	{attribute 'TcIecLibraryType'}
	{attribute 'external_name' := 'F_VN_GradeDataMatrixCodeExp_GUID_48B47258_A931_D3A4_9456_254A5AD23142'}
	(* Grades a Data Matrix code (ECC200) according to ISO / IEC 15415:2011. Requires uniform illumination, good focus and the image sensor plane parallel to the code plane to achieve meaningful results. (expert function) *)
	FUNCTION F_VN_GradeDataMatrixCodeExp : HRESULT
	VAR_INPUT
		ipSrcImage	:	ITcVnImage;	(* Source image, only containing the Data Matrix code region (USINT, 1 channel, including quiet zone) *)
		ipDecodedData	:	REFERENCE TO ITcVnContainer;	(* Returns the decoded data (ContainerType_String_SINT) *)
	END_VAR
	VAR_IN_OUT
		stCodeGrades	:	TcVnCodeGradesDM;	(* Returns the code grades in the range from 0 (very bad) to 4 (very good) *)
	END_VAR
	VAR_INPUT
		fModuleWidth	:	REAL;	(* Minimum module width of the code in the image (in pixels). Must be at least 3, preferably 5 - 8. *)
		ipResultVisualization	:	REFERENCE TO ITcVnImage;	(* Returns a visualization of the scan grid (optional, set to 0 if not required). Module margin grades are color coded: >= 3 as green, >= 2 as light blue, >= 1 as orange, < 1 as red *)
		ipMarginGrades	:	REFERENCE TO ITcVnContainer;	(* Returns the individual margin grade for each module, e.g. to create a custom visualization (optional, set to 0 if not required; ContainerType_Vector_TcVnVector3_REAL, containing [x-position, y-position, grade]) *)
		ipContour	:	REFERENCE TO ITcVnContainer;	(* Returns the 4 code corner points, excluding the quiet zone (optional, set to 0 if not required; ContainerType_Vector_TcVnPoint2_DINT) *)
		hrPrev	:	HRESULT;	(* HRESULT indicating the result of previous operations (If SUCCEEDED(hrPrev) equals false, no operation is executed.) *)
	END_VAR
	VAR_OUTPUT
		fAngleDeg	:	REAL;	(* Returns the clockwise rotation angle in degree *)
	END_VAR

END_FUNCTION

// Functions/Code Quality/F_VN_GradeQRCode

	{attribute 'TcIecLibraryType'}
	{attribute 'external_name' := 'F_VN_GradeQRCode_GUID_2796A0BC_8AD9_DF0A_A63B_3634863F0828'}
	(* Grades a QR code according to ISO / IEC 15415:2011. Requires uniform illumination, good focus and the image sensor plane parallel to the code plane to achieve meaningful results. *)
	FUNCTION F_VN_GradeQRCode : HRESULT
	VAR_INPUT
		ipSrcImage	:	ITcVnImage;	(* Source image, only containing the QR code region (USINT, 1 channel, including quiet zone) *)
		ipDecodedData	:	REFERENCE TO ITcVnContainer;	(* Returns the decoded data (ContainerType_String_SINT) *)
	END_VAR
	VAR_IN_OUT
		stCodeGrades	:	TcVnCodeGradesQR;	(* Returns the code grades in the range from 0 (very bad) to 4 (very good) *)
	END_VAR
	VAR_INPUT
		fModuleWidth	:	REAL;	(* Minimum module width of the code in the image (in pixels). Must be at least 3, preferably 5 - 8. *)
		hrPrev	:	HRESULT;	(* HRESULT indicating the result of previous operations (If SUCCEEDED(hrPrev) equals false, no operation is executed.) *)
	END_VAR
	VAR_OUTPUT
		fAngleDeg	:	REAL;	(* Returns the clockwise rotation angle in degree *)
	END_VAR

END_FUNCTION

// Functions/Code Quality/F_VN_GradeQRCodeExp

	{attribute 'TcIecLibraryType'}
	{attribute 'external_name' := 'F_VN_GradeQRCodeExp_GUID_748E667E_FDFB_D812_893A_DF121E555FAA'}
	(* Grades a QR code according to ISO / IEC 15415:2011. Requires uniform illumination, good focus and the image sensor plane parallel to the code plane to achieve meaningful results. (expert function) *)
	FUNCTION F_VN_GradeQRCodeExp : HRESULT
	VAR_INPUT
		ipSrcImage	:	ITcVnImage;	(* Source image, only containing the QR code region (USINT, 1 channel, including quiet zone) *)
		ipDecodedData	:	REFERENCE TO ITcVnContainer;	(* Returns the decoded data (ContainerType_String_SINT) *)
	END_VAR
	VAR_IN_OUT
		stCodeGrades	:	TcVnCodeGradesQR;	(* Returns the code grades in the range from 0 (very bad) to 4 (very good) *)
	END_VAR
	VAR_INPUT
		fModuleWidth	:	REAL;	(* Minimum module width of the code in the image (in pixels). Must be at least 3, preferably 5 - 8. *)
		ipResultVisualization	:	REFERENCE TO ITcVnImage;	(* Returns a visualization of the scan grid (optional, set to 0 if not required). Module margin grades are color coded: >= 3 as green, >= 2 as light blue, >= 1 as orange, < 1 as red *)
		ipMarginGrades	:	REFERENCE TO ITcVnContainer;	(* Returns the individual margin grade for each module, e.g. to create a custom visualization (optional, set to 0 if not required; ContainerType_Vector_TcVnVector3_REAL, containing [x-position, y-position, grade]) *)
		ipContour	:	REFERENCE TO ITcVnContainer;	(* Returns the 4 code corner points, excluding the quiet zone (optional, set to 0 if not required; ContainerType_Vector_TcVnPoint2_DINT) *)
		hrPrev	:	HRESULT;	(* HRESULT indicating the result of previous operations (If SUCCEEDED(hrPrev) equals false, no operation is executed.) *)
	END_VAR
	VAR_OUTPUT
		fAngleDeg	:	REAL;	(* Returns the clockwise rotation angle in degree *)
	END_VAR

END_FUNCTION

// Functions/Texture Analysis/F_VN_Granulometry

	{attribute 'TcIecLibraryType'}
	{attribute 'external_name' := 'F_VN_Granulometry_GUID_ED4C52B4_5143_D78F_B20E_04305B4C8FA0'}
	(* Computes the granulometry of a textured image using morphological operations. *)
	FUNCTION F_VN_Granulometry : HRESULT
	VAR_INPUT
		ipImage	:	ITcVnImage;	(* Source image (1 channel) *)
		ipIntensityDiffs	:	REFERENCE TO ITcVnContainer;	(* Returns the intensity differences between successive structuring element sizes (CTcVnContainer_Vector_LREAL), which can be used as features for texture description. *)
		eMorphType	:	ETcVnMorphologicalOperator;	(* Only opening or closing are supported. *)
		nMinSize	:	UDINT;	(* Min structuring element size (odd, >= 3) *)
		nMaxSize	:	UDINT;	(* Max structuring element size (>= nMinSize) *)
		nStep	:	UDINT;	(* Step, by which nMinSize is incremented until nMaxSize is exceeded (even, >= 2). *)
		hrPrev	:	HRESULT;	(* HRESULT indicating the result of previous operations (If SUCCEEDED(hrPrev) equals false, no operation is executed.) *)
	END_VAR

END_FUNCTION

// Functions/Texture Analysis/F_VN_HaralickFeatures

	{attribute 'TcIecLibraryType'}
	{attribute 'external_name' := 'F_VN_HaralickFeatures_GUID_C04B3742_2975_D01D_971B_239AA26ADB64'}
	(* Computes the Haralick features of a graylevel image, which describe the texture. *)
	FUNCTION F_VN_HaralickFeatures : HRESULT
	VAR_INPUT
		ipImage	:	ITcVnImage;	(* Source image (1 channel, USINT) *)
		ipFeatures	:	REFERENCE TO ITcVnContainer;	(* Returns the computed Haralick features (CTcVnContainer_Vector_LREAL). The returned feature set contains the mean and standard deviation for each of the first 13 Haralick features, computed for 0, 45, 90, 135 degrees. So there will be 26 features in total (f1 mean, f1 stdDev, f2 mean, f2 stdDev, ..., f13 mean, f13 stdDev). *)
		nDist	:	UDINT;	(* Distance *)
		hrPrev	:	HRESULT;	(* HRESULT indicating the result of previous operations (If SUCCEEDED(hrPrev) equals false, no operation is executed.) *)
	END_VAR

END_FUNCTION

// Functions/OCR/F_VN_OCR

	{attribute 'TcIecLibraryType'}
	{attribute 'external_name' := 'F_VN_OCR_GUID_4649D880_E3A0_D7D8_A83C_DD423A1D4FD0'}
	(* Detects and recognizes characters in a binary image (white characters on black background). *)
	FUNCTION F_VN_OCR : HRESULT
	VAR_INPUT
		ipSrcImage	:	ITcVnImage;	(* Source image (USINT, 1 channel, binary) *)
		eModel	:	ULINT;	(* Selection of OCR model types (ETcVnOcrModelType) *)
		ipCharacters	:	REFERENCE TO ITcVnContainer;	(* Returns the recognized characters (ContainerType_Vector_String_SINT) *)
		hrPrev	:	HRESULT;	(* HRESULT indicating the result of previous operations (If SUCCEEDED(hrPrev) equals false, no operation is executed.) *)
	END_VAR

END_FUNCTION

// Functions/OCR/F_VN_OCRExp

	{attribute 'TcIecLibraryType'}
	{attribute 'external_name' := 'F_VN_OCRExp_GUID_EDBCFF98_0425_D60E_8A16_A0CDB823D474'}
	(* Detects and recognizes characters in a binary image (white characters on black background). (expert function) *)
	FUNCTION F_VN_OCRExp : HRESULT
	VAR_INPUT
		ipSrcImage	:	ITcVnImage;	(* Source image (USINT, 1 channel, binary) *)
		eModel	:	ULINT;	(* Selection of OCR model types (ETcVnOcrModelType) *)
		ipCharacters	:	REFERENCE TO ITcVnContainer;	(* Returns the recognized characters (ContainerType_Vector_String_SINT) *)
	END_VAR
	VAR_IN_OUT CONSTANT
		sPattern	:	STRING;	(* String pattern containing the format in which characters are presented *)
	END_VAR
	VAR_INPUT
		eOcrOptions	:	UDINT;	(* Specifies which options must be applied to the function (ETcVnOcrOptions) *)
		ipBoundingBoxes	:	REFERENCE TO ITcVnContainer;	(* Returns the corresponding bounding boxes of the recognized characters (ContainerType_Vector_TcVnRectangle_DINT, optional, set to 0 if not required) *)
		ipConfidences	:	REFERENCE TO ITcVnContainer;	(* Returns the corresponding classification confidences of the recognized characters (ContainerType_Vector_REAL, optional, set to 0 if not required) *)
		hrPrev	:	HRESULT;	(* HRESULT indicating the result of previous operations (If SUCCEEDED(hrPrev) equals false, no operation is executed.) *)
	END_VAR
	VAR_OUTPUT
		fMinConfidence	:	REAL;	(* Returns the minimum value of the confidences *)
	END_VAR

END_FUNCTION

// Functions/Code Reading/F_VN_ReadBarcode

	{attribute 'TcIecLibraryType'}
	{attribute 'external_name' := 'F_VN_ReadBarcode_GUID_8D55FBD2_3F12_DDCC_85AA_97D1643DAA8D'}
	(* Detect and interpret a 1d barcode within the provided image.
          Can be canceled by Watchdog. *)
	FUNCTION F_VN_ReadBarcode : HRESULT
	VAR_INPUT
		ipSrcImage	:	ITcVnImage;	(* Source image (USINT elements, 1 channel or 3 channel (3 channel input is expected to be RGB and internally converted to Gray)) *)
		ipDecodedData	:	REFERENCE TO ITcVnContainer;	(* Returns the decoded code (ContainerType_Vector_String_SINT) *)
		eBarcodeType	:	UDINT;	(* Types of barcode to search for (ETcVnBarcodeType) *)
		hrPrev	:	HRESULT;	(* HRESULT indicating the result of previous operations (If SUCCEEDED(hrPrev) equals false, no operation is executed.) *)
	END_VAR

END_FUNCTION

// Functions/Code Reading/F_VN_ReadBarcodeExp

	{attribute 'TcIecLibraryType'}
	{attribute 'external_name' := 'F_VN_ReadBarcodeExp_GUID_87DB6D69_2E8D_D7F0_B75F_5C174E4C943E'}
	(* Detect and interpret a 1d barcode within the provided image.
          Can be canceled by Watchdog. *)
	FUNCTION F_VN_ReadBarcodeExp : HRESULT
	VAR_INPUT
		ipSrcImage	:	ITcVnImage;	(* Source image (USINT elements, 1 channel or 3 channel (3 channel input is expected to be RGB and internally converted to Gray)) *)
		ipDecodedData	:	REFERENCE TO ITcVnContainer;	(* Returns the decoded code (ContainerType_Vector_String_SINT) *)
		ipContours	:	REFERENCE TO ITcVnContainer;	(* Returns the code positions as contours (optional, set to 0 if not required; ContainerType_Vector_Vector_TcVnPoint2_DINT) *)
		eBarcodeType	:	UDINT;	(* Types of barcode to search for (ETcVnBarcodeType) *)
		nCodeNumber	:	DINT;	(* Number of 1d barcode that should be detected within the provided image (currently only 1 supported). *)
		eSearchDirection	:	ETcVnBarcodeSearchDirection;	(* Barcode search direction. *)
		hrPrev	:	HRESULT;	(* HRESULT indicating the result of previous operations (If SUCCEEDED(hrPrev) equals false, no operation is executed.) *)
	END_VAR

END_FUNCTION

// Functions/Code Reading/F_VN_ReadBarcodeExp2

	{attribute 'TcIecLibraryType'}
	{attribute 'external_name' := 'F_VN_ReadBarcodeExp2_GUID_4618271E_EA04_D10D_9C61_0BE9FDD29DE9'}
	(* Detect and interpret a 1d barcode within the provided image.
          Can be canceled by Watchdog. *)
	FUNCTION F_VN_ReadBarcodeExp2 : HRESULT
	VAR_INPUT
		ipSrcImage	:	ITcVnImage;	(* Source image (USINT elements, 1 channel or 3 channel (3 channel input is expected to be RGB and internally converted to Gray)) *)
		ipDecodedData	:	REFERENCE TO ITcVnContainer;	(* Returns the decoded code (ContainerType_Vector_String_SINT) *)
		ipContours	:	REFERENCE TO ITcVnContainer;	(* Returns the code positions as contours (optional, set to 0 if not required; ContainerType_Vector_Vector_TcVnPoint2_DINT) *)
		eBarcodeType	:	UDINT;	(* Types of barcode to search for (ETcVnBarcodeType) *)
		nCodeNumber	:	DINT;	(* Number of 1d barcode that should be detected within the provided image (currently only 1 supported). *)
		eSearchDirection	:	ETcVnBarcodeSearchDirection;	(* Barcode search direction. *)
		ipAngles	:	REFERENCE TO ITcVnContainer;	(* Returns the clockwise code rotation angles (optional, set to 0 if not required; ContainerType_Vector_REAL) *)
		hrPrev	:	HRESULT;	(* HRESULT indicating the result of previous operations (If SUCCEEDED(hrPrev) equals false, no operation is executed.) *)
	END_VAR

END_FUNCTION

// Functions/Code Reading/F_VN_ReadDataMatrixCode

	{attribute 'TcIecLibraryType'}
	{attribute 'external_name' := 'F_VN_ReadDataMatrixCode_GUID_47E4E701_DDFF_D5D8_A6D3_EAF32B974F2E'}
	(* Detect and interpret a data matrix code (ECC200) within the provided image. *)
	FUNCTION F_VN_ReadDataMatrixCode : HRESULT
	VAR_INPUT
		ipSrcImage	:	ITcVnImage;	(* Source image (USINT elements, 1 or 3 channels) *)
		ipDecodedData	:	REFERENCE TO ITcVnContainer;	(* Returns the decoded code (ContainerType_Vector_String_SINT) *)
		hrPrev	:	HRESULT;	(* HRESULT indicating the result of previous operations (If SUCCEEDED(hrPrev) equals false, no operation is executed.) *)
	END_VAR

END_FUNCTION

// Functions/Code Reading/F_VN_ReadDataMatrixCodeExp

	{attribute 'TcIecLibraryType'}
	{attribute 'external_name' := 'F_VN_ReadDataMatrixCodeExp_GUID_D9BF17C7_F534_DAB1_8EBB_28E139EC8F96'}
	(* Detect and interpret a data matrix code (ECC200) within the provided image. *)
	FUNCTION F_VN_ReadDataMatrixCodeExp : HRESULT
	VAR_INPUT
		ipSrcImage	:	ITcVnImage;	(* Source image (USINT elements, 1 or 3 channels) *)
		ipDecodedData	:	REFERENCE TO ITcVnContainer;	(* Returns the decoded code (ContainerType_Vector_String_SINT) *)
		ipContours	:	REFERENCE TO ITcVnContainer;	(* Returns the code positions as contours (optional, set to 0 if not required; ContainerType_Vector_Vector_TcVnPoint2_DINT) *)
		nCodeNumber	:	DINT;	(* Number of data matrix codes that should be detected within the provided image. (If set to -1, it tries to detect all data matrix codes.) *)
		eSearchStrategy	:	UDINT;	(* Used search strategy (ETcVn2dCodeSearchStrategy) *)
		hrPrev	:	HRESULT;	(* HRESULT indicating the result of previous operations (If SUCCEEDED(hrPrev) equals false, no operation is executed.) *)
	END_VAR

END_FUNCTION

// Functions/Code Reading/F_VN_ReadDataMatrixCodeExp2

	{attribute 'TcIecLibraryType'}
	{attribute 'external_name' := 'F_VN_ReadDataMatrixCodeExp2_GUID_09005C2B_5490_D76C_85BF_2B9D22242AE9'}
	(* Detect and interpret a data matrix code (ECC200) within the provided image. *)
	FUNCTION F_VN_ReadDataMatrixCodeExp2 : HRESULT
	VAR_INPUT
		ipSrcImage	:	ITcVnImage;	(* Source image (USINT elements, 1 or 3 channels) *)
		ipDecodedData	:	REFERENCE TO ITcVnContainer;	(* Returns the decoded code (ContainerType_Vector_String_SINT) *)
		ipContours	:	REFERENCE TO ITcVnContainer;	(* Returns the code positions as contours (optional, set to 0 if not required; ContainerType_Vector_Vector_TcVnPoint2_DINT) *)
		nCodeNumber	:	DINT;	(* Number of data matrix codes that should be detected within the provided image. (If set to -1, it tries to detect all data matrix codes.) *)
		eSearchStrategy	:	UDINT;	(* Used search strategy (ETcVn2dCodeSearchStrategy) *)
		ipAngles	:	REFERENCE TO ITcVnContainer;	(* Returns the clockwise code rotation angles (optional, set to 0 if not required; ContainerType_Vector_REAL) *)
		hrPrev	:	HRESULT;	(* HRESULT indicating the result of previous operations (If SUCCEEDED(hrPrev) equals false, no operation is executed.) *)
	END_VAR

END_FUNCTION

// Functions/Code Reading/F_VN_ReadDataMatrixCodeRoi

	{attribute 'TcIecLibraryType'}
	{attribute 'external_name' := 'F_VN_ReadDataMatrixCodeRoi_GUID_48E5E96D_F4D5_D058_B628_BE3202493787'}
	(* Detect and interpret a data matrix code (ECC200) within the provided image. The code should be in the image center. *)
	FUNCTION F_VN_ReadDataMatrixCodeRoi : HRESULT
	VAR_INPUT
		ipSrcImage	:	ITcVnImage;	(* Source image (USINT elements, 1 channel) *)
		ipDecodedData	:	REFERENCE TO ITcVnContainer;	(* Returns the decoded code (ContainerType_String_SINT) *)
		fModuleWidth	:	REAL;	(* Minimum module width of the code in the image (in pixels). Must be at least 3, preferably 5 - 8. *)
		hrPrev	:	HRESULT;	(* HRESULT indicating the result of previous operations (If SUCCEEDED(hrPrev) equals false, no operation is executed.) *)
	END_VAR
	VAR_OUTPUT
		fAngleDeg	:	REAL;	(* Returns the clockwise rotation angle in degree *)
	END_VAR

END_FUNCTION

// Functions/Code Reading/F_VN_ReadDataMatrixCodeRoiExp

	{attribute 'TcIecLibraryType'}
	{attribute 'external_name' := 'F_VN_ReadDataMatrixCodeRoiExp_GUID_46D2D5C0_3E23_D29F_BAD8_6FE587ABCD92'}
	(* Detect and interpret a data matrix code (ECC200) within the provided image. The code should be in the image center. (expert function) *)
	FUNCTION F_VN_ReadDataMatrixCodeRoiExp : HRESULT
	VAR_INPUT
		ipSrcImage	:	ITcVnImage;	(* Source image (USINT elements, 1 channel) *)
		ipDecodedData	:	REFERENCE TO ITcVnContainer;	(* Returns the decoded code (ContainerType_String_SINT) *)
		fModuleWidth	:	REAL;	(* Minimum module width of the code in the image (in pixels). Must be at least 3, preferably 5 - 8. *)
		ipContour	:	REFERENCE TO ITcVnContainer;	(* Returns the contour of the detected code (ContainerType_Vector_TcVnPoint2_DINT; optional, set to 0 if not required) *)
		eOptions	:	ULINT;	(* Specifies a combination of one or more ETcVnDataMatrixOptions *)
		nRows	:	USINT;	(* Specifies the number of code module rows, including the finder and clock pattern, excluding the quiet zone (8 - 144; set to 0 to search for any size) *)
		nCols	:	USINT;	(* Specifies the number of code module columns, including the finder and clock pattern, excluding the quiet zone (10 - 144; set to 0 to search for any size) *)
		bExtensiveSearch	:	BOOL;	(* If true, tries different approaches if the specified options fail *)
		hrPrev	:	HRESULT;	(* HRESULT indicating the result of previous operations (If SUCCEEDED(hrPrev) equals false, no operation is executed.) *)
	END_VAR
	VAR_OUTPUT
		fAngleDeg	:	REAL;	(* Returns the clockwise rotation angle in degree *)
	END_VAR

END_FUNCTION

// Functions/Code Reading/F_VN_ReadPharmaCode

	{attribute 'TcIecLibraryType'}
	{attribute 'external_name' := 'F_VN_ReadPharmaCode_GUID_1552A435_B815_D86A_80F6_32509F0D267A'}
	(* Detect and interpret a pharma code within the provided image.
				Can be canceled by Watchdog. *)
	FUNCTION F_VN_ReadPharmaCode : HRESULT
	VAR_INPUT
		ipSrcImage	:	ITcVnImage;	(* Source image (1 channel (all element types) or 3 channel with elements of type TCVN_ET_USINT, TCVN_ET_UINT or TCVN_ET_REAL (3 channel input is expected to be RGB and internally converted to Gray)) *)
		ipDecodedData	:	REFERENCE TO ITcVnContainer;	(* Returns the decoded code (ContainerType_Vector_String_SINT) *)
		hrPrev	:	HRESULT;	(* HRESULT indicating the result of previous operations (If SUCCEEDED(hrPrev) equals false, no operation is executed.) *)
	END_VAR

END_FUNCTION

// Functions/Code Reading/F_VN_ReadPharmaCodeExp

	{attribute 'TcIecLibraryType'}
	{attribute 'external_name' := 'F_VN_ReadPharmaCodeExp_GUID_104C8116_6161_DF69_8F4B_5E4188AB2031'}
	(* Detect and interpret a pharma code within the provided image.
				Can be canceled by Watchdog. *)
	FUNCTION F_VN_ReadPharmaCodeExp : HRESULT
	VAR_INPUT
		ipSrcImage	:	ITcVnImage;	(* Source image (1 channel (all element types) or 3 channel with elements of type TCVN_ET_USINT, TCVN_ET_UINT or TCVN_ET_REAL (3 channel input is expected to be RGB and internally converted to Gray)) *)
		ipDecodedData	:	REFERENCE TO ITcVnContainer;	(* Returns the decoded code (ContainerType_Vector_String_SINT) *)
		ipContours	:	REFERENCE TO ITcVnContainer;	(* Returns the code positions as contours (optional, set to 0 if not required; ContainerType_Vector_Vector_TcVnPoint2_DINT) *)
		nCodeNumber	:	DINT;	(* Number of pharma codes that should be detected within the provided image (currently only 1 supported). *)
		nMinBarNumber	:	INT;	(* Minimal number of (dark) bars that codes must have. *)
		hrPrev	:	HRESULT;	(* HRESULT indicating the result of previous operations (If SUCCEEDED(hrPrev) equals false, no operation is executed.) *)
	END_VAR

END_FUNCTION

// Functions/Code Reading/F_VN_ReadPharmaCodeExp2

	{attribute 'TcIecLibraryType'}
	{attribute 'external_name' := 'F_VN_ReadPharmaCodeExp2_GUID_9680F0AE_00B1_D565_BEF4_E7C60C82665F'}
	(* Detect and interpret a pharma code within the provided image.
				Can be canceled by Watchdog. *)
	FUNCTION F_VN_ReadPharmaCodeExp2 : HRESULT
	VAR_INPUT
		ipSrcImage	:	ITcVnImage;	(* Source image (1 channel (all element types) or 3 channel with elements of type TCVN_ET_USINT, TCVN_ET_UINT or TCVN_ET_REAL (3 channel input is expected to be RGB and internally converted to Gray)) *)
		ipDecodedData	:	REFERENCE TO ITcVnContainer;	(* Returns the decoded code (ContainerType_Vector_String_SINT) *)
		ipContours	:	REFERENCE TO ITcVnContainer;	(* Returns the code positions as contours (optional, set to 0 if not required; ContainerType_Vector_Vector_TcVnPoint2_DINT) *)
		nCodeNumber	:	DINT;	(* Number of pharma codes that should be detected within the provided image (currently only 1 supported). *)
		nMinBarNumber	:	INT;	(* Minimal number of (dark) bars that codes must have. *)
		ipAngles	:	REFERENCE TO ITcVnContainer;	(* Returns the clockwise code rotation angles (optional, set to 0 if not required; ContainerType_Vector_REAL) *)
		hrPrev	:	HRESULT;	(* HRESULT indicating the result of previous operations (If SUCCEEDED(hrPrev) equals false, no operation is executed.) *)
	END_VAR

END_FUNCTION

// Functions/Code Reading/F_VN_ReadQRCode

	{attribute 'TcIecLibraryType'}
	{attribute 'external_name' := 'F_VN_ReadQRCode_GUID_920DC6C0_AA3D_D3AA_AB2C_E13D9C544BB8'}
	(* Detect and interpret a QR code within the provided image.
          Can be canceled by Watchdog. *)
	FUNCTION F_VN_ReadQRCode : HRESULT
	VAR_INPUT
		ipSrcImage	:	ITcVnImage;	(* Source image (USINT elements, 1 channel or 3 channel (3 channel input is expected to be RGB and internally converted to Gray)) *)
		ipDecodedData	:	REFERENCE TO ITcVnContainer;	(* Returns the decoded code (ContainerType_Vector_String_SINT) *)
		hrPrev	:	HRESULT;	(* HRESULT indicating the result of previous operations (If SUCCEEDED(hrPrev) equals false, no operation is executed.) *)
	END_VAR

END_FUNCTION

// Functions/Code Reading/F_VN_ReadQRCodeExp

	{attribute 'TcIecLibraryType'}
	{attribute 'external_name' := 'F_VN_ReadQRCodeExp_GUID_1FBD3D65_B71B_D593_A041_BAEB18B892EA'}
	(* Detect and interpret a QR code within the provided image.
          Can be canceled by Watchdog. *)
	FUNCTION F_VN_ReadQRCodeExp : HRESULT
	VAR_INPUT
		ipSrcImage	:	ITcVnImage;	(* Source image (USINT elements, 1 channel or 3 channel (3 channel input is expected to be RGB and internally converted to Gray)) *)
		ipDecodedData	:	REFERENCE TO ITcVnContainer;	(* Returns the decoded code (ContainerType_Vector_String_SINT) *)
		ipContours	:	REFERENCE TO ITcVnContainer;	(* Returns the code positions as contours (optional, set to 0 if not required; ContainerType_Vector_Vector_TcVnPoint2_DINT) *)
		nCodeNumber	:	DINT;	(* Number of QR codes that should be detected within the provided image (currently only 1 supported). *)
		eSearchStrategy	:	UDINT;	(* Used search strategy (ETcVn2dCodeSearchStrategy) *)
		hrPrev	:	HRESULT;	(* HRESULT indicating the result of previous operations (If SUCCEEDED(hrPrev) equals false, no operation is executed.) *)
	END_VAR

END_FUNCTION

// Functions/Code Reading/F_VN_ReadQRCodeExp2

	{attribute 'TcIecLibraryType'}
	{attribute 'external_name' := 'F_VN_ReadQRCodeExp2_GUID_3AB569A0_9D43_DE15_9C74_8765ADC435B0'}
	(* Detect and interpret a QR code within the provided image.
          Can be canceled by Watchdog. *)
	FUNCTION F_VN_ReadQRCodeExp2 : HRESULT
	VAR_INPUT
		ipSrcImage	:	ITcVnImage;	(* Source image (USINT elements, 1 channel or 3 channel (3 channel input is expected to be RGB and internally converted to Gray)) *)
		ipDecodedData	:	REFERENCE TO ITcVnContainer;	(* Returns the decoded code (ContainerType_Vector_String_SINT) *)
		ipContours	:	REFERENCE TO ITcVnContainer;	(* Returns the code positions as contours (optional, set to 0 if not required; ContainerType_Vector_Vector_TcVnPoint2_DINT) *)
		nCodeNumber	:	DINT;	(* Number of QR codes that should be detected within the provided image (currently only 1 supported). *)
		eSearchStrategy	:	UDINT;	(* Used search strategy (ETcVn2dCodeSearchStrategy) *)
		ipAngles	:	REFERENCE TO ITcVnContainer;	(* Returns the clockwise code rotation angles (optional, set to 0 if not required; ContainerType_Vector_REAL) *)
		hrPrev	:	HRESULT;	(* HRESULT indicating the result of previous operations (If SUCCEEDED(hrPrev) equals false, no operation is executed.) *)
	END_VAR

END_FUNCTION

// Functions/Algebraic Container Operations/F_VN_AddToContainerElements/F_VN_AddToContainerElements_DINT

	{attribute 'TcIecLibraryType'}
	{attribute 'external_name' := 'F_VN_AddToContainerElements_DINT_GUID_343313F6_A496_DC3B_B1B9_388E62CB725C'}
	(* Add a value to each container element. *)
	FUNCTION F_VN_AddToContainerElements_DINT : HRESULT
	VAR_INPUT
		nValue	:	DINT;	(* Value *)
		ipContainer	:	ITcVnContainer;	(* Container with DINT elements *)
		hrPrev	:	HRESULT;	(* HRESULT indicating the result of previous operations (If SUCCEEDED(hrPrev) equals false, no operation is executed.) *)
	END_VAR

END_FUNCTION

// Functions/Algebraic Container Operations/F_VN_AddToContainerElements/F_VN_AddToContainerElements_INT

	{attribute 'TcIecLibraryType'}
	{attribute 'external_name' := 'F_VN_AddToContainerElements_INT_GUID_E9C6EA43_ACCF_DEFB_9BF4_897C0F2FC8FA'}
	(* Add a value to each container element. *)
	FUNCTION F_VN_AddToContainerElements_INT : HRESULT
	VAR_INPUT
		nValue	:	INT;	(* Value *)
		ipContainer	:	ITcVnContainer;	(* Container with INT elements *)
		hrPrev	:	HRESULT;	(* HRESULT indicating the result of previous operations (If SUCCEEDED(hrPrev) equals false, no operation is executed.) *)
	END_VAR

END_FUNCTION

// Functions/Algebraic Container Operations/F_VN_AddToContainerElements/F_VN_AddToContainerElements_LREAL

	{attribute 'TcIecLibraryType'}
	{attribute 'external_name' := 'F_VN_AddToContainerElements_LREAL_GUID_8BBAD9B2_A422_DA40_8842_E5469A52D3D0'}
	(* Add a value to each container element. *)
	FUNCTION F_VN_AddToContainerElements_LREAL : HRESULT
	VAR_INPUT
		fValue	:	LREAL;	(* Value *)
		ipContainer	:	ITcVnContainer;	(* Container with LREAL elements *)
		hrPrev	:	HRESULT;	(* HRESULT indicating the result of previous operations (If SUCCEEDED(hrPrev) equals false, no operation is executed.) *)
	END_VAR

END_FUNCTION

// Functions/Algebraic Container Operations/F_VN_AddToContainerElements/F_VN_AddToContainerElements_REAL

	{attribute 'TcIecLibraryType'}
	{attribute 'external_name' := 'F_VN_AddToContainerElements_REAL_GUID_068D7646_CFE3_D05D_9927_0097B5790E16'}
	(* Add a value to each container element. *)
	FUNCTION F_VN_AddToContainerElements_REAL : HRESULT
	VAR_INPUT
		fValue	:	REAL;	(* Value *)
		ipContainer	:	ITcVnContainer;	(* Container with REAL elements *)
		hrPrev	:	HRESULT;	(* HRESULT indicating the result of previous operations (If SUCCEEDED(hrPrev) equals false, no operation is executed.) *)
	END_VAR

END_FUNCTION

// Functions/Algebraic Container Operations/F_VN_AddToContainerElements/F_VN_AddToContainerElements_SINT

	{attribute 'TcIecLibraryType'}
	{attribute 'external_name' := 'F_VN_AddToContainerElements_SINT_GUID_4DCFF384_F53F_D449_9B15_671331675EFE'}
	(* Add a value to each container element. *)
	FUNCTION F_VN_AddToContainerElements_SINT : HRESULT
	VAR_INPUT
		nValue	:	SINT;	(* Value *)
		ipContainer	:	ITcVnContainer;	(* Container with SINT elements *)
		hrPrev	:	HRESULT;	(* HRESULT indicating the result of previous operations (If SUCCEEDED(hrPrev) equals false, no operation is executed.) *)
	END_VAR

END_FUNCTION

// Functions/Algebraic Container Operations/F_VN_AddToContainerElements/F_VN_AddToContainerElements_TcVnKeyPoint

	{attribute 'TcIecLibraryType'}
	{attribute 'external_name' := 'F_VN_AddToContainerElements_TcVnKeyPoint_GUID_54FF73F9_C73B_D4F0_B6FA_FD4148B8A9D6'}
	(* Add a value to each container element. *)
	FUNCTION F_VN_AddToContainerElements_TcVnKeyPoint : HRESULT
	VAR_IN_OUT
		stValue	:	TcVnKeyPoint;	(* Value *)
	END_VAR
	VAR_INPUT
		ipContainer	:	ITcVnContainer;	(* Container with TcVnKeyPoint elements *)
		hrPrev	:	HRESULT;	(* HRESULT indicating the result of previous operations (If SUCCEEDED(hrPrev) equals false, no operation is executed.) *)
	END_VAR

END_FUNCTION

// Functions/Algebraic Container Operations/F_VN_AddToContainerElements/F_VN_AddToContainerElements_TcVnPoint2_DINT

	{attribute 'TcIecLibraryType'}
	{attribute 'external_name' := 'F_VN_AddToContainerElements_TcVnPoint2_DINT_GUID_6E237BBA_4475_D7AD_8453_E663E04986A0'}
	(* Add a value to each container element. *)
	FUNCTION F_VN_AddToContainerElements_TcVnPoint2_DINT : HRESULT
	VAR_IN_OUT
		aValue	:	TcVnPoint2_DINT;	(* Value *)
	END_VAR
	VAR_INPUT
		ipContainer	:	ITcVnContainer;	(* Container with TcVnPoint2_DINT elements *)
		hrPrev	:	HRESULT;	(* HRESULT indicating the result of previous operations (If SUCCEEDED(hrPrev) equals false, no operation is executed.) *)
	END_VAR

END_FUNCTION

// Functions/Algebraic Container Operations/F_VN_AddToContainerElements/F_VN_AddToContainerElements_TcVnPoint2_LREAL

	{attribute 'TcIecLibraryType'}
	{attribute 'external_name' := 'F_VN_AddToContainerElements_TcVnPoint2_LREAL_GUID_2CD023F6_4D8E_D476_BA0F_795BA163BD7B'}
	(* Add a value to each container element. *)
	FUNCTION F_VN_AddToContainerElements_TcVnPoint2_LREAL : HRESULT
	VAR_IN_OUT
		aValue	:	TcVnPoint2_LREAL;	(* Value *)
	END_VAR
	VAR_INPUT
		ipContainer	:	ITcVnContainer;	(* Container with TcVnPoint2_LREAL elements *)
		hrPrev	:	HRESULT;	(* HRESULT indicating the result of previous operations (If SUCCEEDED(hrPrev) equals false, no operation is executed.) *)
	END_VAR

END_FUNCTION

// Functions/Algebraic Container Operations/F_VN_AddToContainerElements/F_VN_AddToContainerElements_TcVnPoint2_REAL

	{attribute 'TcIecLibraryType'}
	{attribute 'external_name' := 'F_VN_AddToContainerElements_TcVnPoint2_REAL_GUID_6F306FAC_FD53_D78B_8D14_692E0DCBC5AF'}
	(* Add a value to each container element. *)
	FUNCTION F_VN_AddToContainerElements_TcVnPoint2_REAL : HRESULT
	VAR_IN_OUT
		aValue	:	TcVnPoint2_REAL;	(* Value *)
	END_VAR
	VAR_INPUT
		ipContainer	:	ITcVnContainer;	(* Container with TcVnPoint2_REAL elements *)
		hrPrev	:	HRESULT;	(* HRESULT indicating the result of previous operations (If SUCCEEDED(hrPrev) equals false, no operation is executed.) *)
	END_VAR

END_FUNCTION

// Functions/Algebraic Container Operations/F_VN_AddToContainerElements/F_VN_AddToContainerElements_TcVnPoint3_LREAL

	{attribute 'TcIecLibraryType'}
	{attribute 'external_name' := 'F_VN_AddToContainerElements_TcVnPoint3_LREAL_GUID_EC3D95DD_9FEB_DB86_AFF3_8DEFA5264BA8'}
	(* Add a value to each container element. *)
	FUNCTION F_VN_AddToContainerElements_TcVnPoint3_LREAL : HRESULT
	VAR_IN_OUT
		aValue	:	TcVnPoint3_LREAL;	(* Value *)
	END_VAR
	VAR_INPUT
		ipContainer	:	ITcVnContainer;	(* Container with TcVnPoint3_LREAL elements *)
		hrPrev	:	HRESULT;	(* HRESULT indicating the result of previous operations (If SUCCEEDED(hrPrev) equals false, no operation is executed.) *)
	END_VAR

END_FUNCTION

// Functions/Algebraic Container Operations/F_VN_AddToContainerElements/F_VN_AddToContainerElements_TcVnPoint3_REAL

	{attribute 'TcIecLibraryType'}
	{attribute 'external_name' := 'F_VN_AddToContainerElements_TcVnPoint3_REAL_GUID_10205EB2_B361_D98B_9995_E1C2C42183E5'}
	(* Add a value to each container element. *)
	FUNCTION F_VN_AddToContainerElements_TcVnPoint3_REAL : HRESULT
	VAR_IN_OUT
		aValue	:	TcVnPoint3_REAL;	(* Value *)
	END_VAR
	VAR_INPUT
		ipContainer	:	ITcVnContainer;	(* Container with TcVnPoint3_REAL elements *)
		hrPrev	:	HRESULT;	(* HRESULT indicating the result of previous operations (If SUCCEEDED(hrPrev) equals false, no operation is executed.) *)
	END_VAR

END_FUNCTION

// Functions/Algebraic Container Operations/F_VN_AddToContainerElements/F_VN_AddToContainerElements_TcVnRectangle_DINT

	{attribute 'TcIecLibraryType'}
	{attribute 'external_name' := 'F_VN_AddToContainerElements_TcVnRectangle_DINT_GUID_38F2D84E_AF00_D872_903F_225627D05641'}
	(* Add a value to each container element. *)
	FUNCTION F_VN_AddToContainerElements_TcVnRectangle_DINT : HRESULT
	VAR_IN_OUT
		stValue	:	TcVnRectangle_DINT;	(* Value *)
	END_VAR
	VAR_INPUT
		ipContainer	:	ITcVnContainer;	(* Container with TcVnRectangle_DINT elements *)
		hrPrev	:	HRESULT;	(* HRESULT indicating the result of previous operations (If SUCCEEDED(hrPrev) equals false, no operation is executed.) *)
	END_VAR

END_FUNCTION

// Functions/Algebraic Container Operations/F_VN_AddToContainerElements/F_VN_AddToContainerElements_TcVnRotatedRectangle

	{attribute 'TcIecLibraryType'}
	{attribute 'external_name' := 'F_VN_AddToContainerElements_TcVnRotatedRectangle_GUID_0BB16037_63BB_DFD9_97D3_D3BDAD492DA6'}
	(* Add a value to each container element. *)
	FUNCTION F_VN_AddToContainerElements_TcVnRotatedRectangle : HRESULT
	VAR_IN_OUT
		stValue	:	TcVnRotatedRectangle;	(* Value *)
	END_VAR
	VAR_INPUT
		ipContainer	:	ITcVnContainer;	(* Container with TcVnRotatedRectangle elements *)
		hrPrev	:	HRESULT;	(* HRESULT indicating the result of previous operations (If SUCCEEDED(hrPrev) equals false, no operation is executed.) *)
	END_VAR

END_FUNCTION

// Functions/Algebraic Container Operations/F_VN_AddToContainerElements/F_VN_AddToContainerElements_TcVnVector2_DINT

	{attribute 'TcIecLibraryType'}
	{attribute 'external_name' := 'F_VN_AddToContainerElements_TcVnVector2_DINT_GUID_92A51B70_5462_DC20_B97B_2B50E16496F5'}
	(* Add a value to each container element. *)
	FUNCTION F_VN_AddToContainerElements_TcVnVector2_DINT : HRESULT
	VAR_IN_OUT
		aValue	:	TcVnVector2_DINT;	(* Value *)
	END_VAR
	VAR_INPUT
		ipContainer	:	ITcVnContainer;	(* Container with TcVnVector2_DINT elements *)
		hrPrev	:	HRESULT;	(* HRESULT indicating the result of previous operations (If SUCCEEDED(hrPrev) equals false, no operation is executed.) *)
	END_VAR

END_FUNCTION

// Functions/Algebraic Container Operations/F_VN_AddToContainerElements/F_VN_AddToContainerElements_TcVnVector2_INT

	{attribute 'TcIecLibraryType'}
	{attribute 'external_name' := 'F_VN_AddToContainerElements_TcVnVector2_INT_GUID_35D96140_D0B0_D245_91B0_11320BB08D28'}
	(* Add a value to each container element. *)
	FUNCTION F_VN_AddToContainerElements_TcVnVector2_INT : HRESULT
	VAR_IN_OUT
		aValue	:	TcVnVector2_INT;	(* Value *)
	END_VAR
	VAR_INPUT
		ipContainer	:	ITcVnContainer;	(* Container with TcVnVector2_INT elements *)
		hrPrev	:	HRESULT;	(* HRESULT indicating the result of previous operations (If SUCCEEDED(hrPrev) equals false, no operation is executed.) *)
	END_VAR

END_FUNCTION

// Functions/Algebraic Container Operations/F_VN_AddToContainerElements/F_VN_AddToContainerElements_TcVnVector2_REAL

	{attribute 'TcIecLibraryType'}
	{attribute 'external_name' := 'F_VN_AddToContainerElements_TcVnVector2_REAL_GUID_77D06AA4_46F9_D084_81E3_88F329576A93'}
	(* Add a value to each container element. *)
	FUNCTION F_VN_AddToContainerElements_TcVnVector2_REAL : HRESULT
	VAR_IN_OUT
		aValue	:	TcVnVector2_REAL;	(* Value *)
	END_VAR
	VAR_INPUT
		ipContainer	:	ITcVnContainer;	(* Container with TcVnVector2_REAL elements *)
		hrPrev	:	HRESULT;	(* HRESULT indicating the result of previous operations (If SUCCEEDED(hrPrev) equals false, no operation is executed.) *)
	END_VAR

END_FUNCTION

// Functions/Algebraic Container Operations/F_VN_AddToContainerElements/F_VN_AddToContainerElements_TcVnVector2_SINT

	{attribute 'TcIecLibraryType'}
	{attribute 'external_name' := 'F_VN_AddToContainerElements_TcVnVector2_SINT_GUID_D5268A60_1337_DEC9_AB62_F835565AE23F'}
	(* Add a value to each container element. *)
	FUNCTION F_VN_AddToContainerElements_TcVnVector2_SINT : HRESULT
	VAR_IN_OUT
		aValue	:	TcVnVector2_SINT;	(* Value *)
	END_VAR
	VAR_INPUT
		ipContainer	:	ITcVnContainer;	(* Container with TcVnVector2_SINT elements *)
		hrPrev	:	HRESULT;	(* HRESULT indicating the result of previous operations (If SUCCEEDED(hrPrev) equals false, no operation is executed.) *)
	END_VAR

END_FUNCTION

// Functions/Algebraic Container Operations/F_VN_AddToContainerElements/F_VN_AddToContainerElements_TcVnVector2_UINT

	{attribute 'TcIecLibraryType'}
	{attribute 'external_name' := 'F_VN_AddToContainerElements_TcVnVector2_UINT_GUID_3995719B_FEF6_DA24_83CF_4EDB4D9BC5D8'}
	(* Add a value to each container element. *)
	FUNCTION F_VN_AddToContainerElements_TcVnVector2_UINT : HRESULT
	VAR_IN_OUT
		aValue	:	TcVnVector2_UINT;	(* Value *)
	END_VAR
	VAR_INPUT
		ipContainer	:	ITcVnContainer;	(* Container with TcVnVector2_UINT elements *)
		hrPrev	:	HRESULT;	(* HRESULT indicating the result of previous operations (If SUCCEEDED(hrPrev) equals false, no operation is executed.) *)
	END_VAR

END_FUNCTION

// Functions/Algebraic Container Operations/F_VN_AddToContainerElements/F_VN_AddToContainerElements_TcVnVector2_USINT

	{attribute 'TcIecLibraryType'}
	{attribute 'external_name' := 'F_VN_AddToContainerElements_TcVnVector2_USINT_GUID_7620B2DD_DC8E_D8AC_9E84_6D7D2520652B'}
	(* Add a value to each container element. *)
	FUNCTION F_VN_AddToContainerElements_TcVnVector2_USINT : HRESULT
	VAR_IN_OUT
		aValue	:	TcVnVector2_USINT;	(* Value *)
	END_VAR
	VAR_INPUT
		ipContainer	:	ITcVnContainer;	(* Container with TcVnVector2_USINT elements *)
		hrPrev	:	HRESULT;	(* HRESULT indicating the result of previous operations (If SUCCEEDED(hrPrev) equals false, no operation is executed.) *)
	END_VAR

END_FUNCTION

// Functions/Algebraic Container Operations/F_VN_AddToContainerElements/F_VN_AddToContainerElements_TcVnVector3_INT

	{attribute 'TcIecLibraryType'}
	{attribute 'external_name' := 'F_VN_AddToContainerElements_TcVnVector3_INT_GUID_1E7C3B0C_DD01_DBBF_9DC0_6429161C8DDB'}
	(* Add a value to each container element. *)
	FUNCTION F_VN_AddToContainerElements_TcVnVector3_INT : HRESULT
	VAR_IN_OUT
		aValue	:	TcVnVector3_INT;	(* Value *)
	END_VAR
	VAR_INPUT
		ipContainer	:	ITcVnContainer;	(* Container with TcVnVector3_INT elements *)
		hrPrev	:	HRESULT;	(* HRESULT indicating the result of previous operations (If SUCCEEDED(hrPrev) equals false, no operation is executed.) *)
	END_VAR

END_FUNCTION

// Functions/Algebraic Container Operations/F_VN_AddToContainerElements/F_VN_AddToContainerElements_TcVnVector3_REAL

	{attribute 'TcIecLibraryType'}
	{attribute 'external_name' := 'F_VN_AddToContainerElements_TcVnVector3_REAL_GUID_680E08F1_52F7_D04D_88A3_EC4C6EF2E4E5'}
	(* Add a value to each container element. *)
	FUNCTION F_VN_AddToContainerElements_TcVnVector3_REAL : HRESULT
	VAR_IN_OUT
		aValue	:	TcVnVector3_REAL;	(* Value *)
	END_VAR
	VAR_INPUT
		ipContainer	:	ITcVnContainer;	(* Container with TcVnVector3_REAL elements *)
		hrPrev	:	HRESULT;	(* HRESULT indicating the result of previous operations (If SUCCEEDED(hrPrev) equals false, no operation is executed.) *)
	END_VAR

END_FUNCTION

// Functions/Algebraic Container Operations/F_VN_AddToContainerElements/F_VN_AddToContainerElements_TcVnVector3_SINT

	{attribute 'TcIecLibraryType'}
	{attribute 'external_name' := 'F_VN_AddToContainerElements_TcVnVector3_SINT_GUID_04FFB0CE_CFFC_D05E_B249_D5DA676AF07B'}
	(* Add a value to each container element. *)
	FUNCTION F_VN_AddToContainerElements_TcVnVector3_SINT : HRESULT
	VAR_IN_OUT
		aValue	:	TcVnVector3_SINT;	(* Value *)
	END_VAR
	VAR_INPUT
		ipContainer	:	ITcVnContainer;	(* Container with TcVnVector3_SINT elements *)
		hrPrev	:	HRESULT;	(* HRESULT indicating the result of previous operations (If SUCCEEDED(hrPrev) equals false, no operation is executed.) *)
	END_VAR

END_FUNCTION

// Functions/Algebraic Container Operations/F_VN_AddToContainerElements/F_VN_AddToContainerElements_TcVnVector3_UINT

	{attribute 'TcIecLibraryType'}
	{attribute 'external_name' := 'F_VN_AddToContainerElements_TcVnVector3_UINT_GUID_AD9A624B_EAD1_DABC_8566_82FDAB24C64E'}
	(* Add a value to each container element. *)
	FUNCTION F_VN_AddToContainerElements_TcVnVector3_UINT : HRESULT
	VAR_IN_OUT
		aValue	:	TcVnVector3_UINT;	(* Value *)
	END_VAR
	VAR_INPUT
		ipContainer	:	ITcVnContainer;	(* Container with TcVnVector3_UINT elements *)
		hrPrev	:	HRESULT;	(* HRESULT indicating the result of previous operations (If SUCCEEDED(hrPrev) equals false, no operation is executed.) *)
	END_VAR

END_FUNCTION

// Functions/Algebraic Container Operations/F_VN_AddToContainerElements/F_VN_AddToContainerElements_TcVnVector3_USINT

	{attribute 'TcIecLibraryType'}
	{attribute 'external_name' := 'F_VN_AddToContainerElements_TcVnVector3_USINT_GUID_B8F25D60_2E70_D6E8_82F2_5D646C75AC8C'}
	(* Add a value to each container element. *)
	FUNCTION F_VN_AddToContainerElements_TcVnVector3_USINT : HRESULT
	VAR_IN_OUT
		aValue	:	TcVnVector3_USINT;	(* Value *)
	END_VAR
	VAR_INPUT
		ipContainer	:	ITcVnContainer;	(* Container with TcVnVector3_USINT elements *)
		hrPrev	:	HRESULT;	(* HRESULT indicating the result of previous operations (If SUCCEEDED(hrPrev) equals false, no operation is executed.) *)
	END_VAR

END_FUNCTION

// Functions/Algebraic Container Operations/F_VN_AddToContainerElements/F_VN_AddToContainerElements_TcVnVector4_DINT

	{attribute 'TcIecLibraryType'}
	{attribute 'external_name' := 'F_VN_AddToContainerElements_TcVnVector4_DINT_GUID_B8E2867C_2EFD_D80B_9C97_55E779F27765'}
	(* Add a value to each container element. *)
	FUNCTION F_VN_AddToContainerElements_TcVnVector4_DINT : HRESULT
	VAR_IN_OUT
		aValue	:	TcVnVector4_DINT;	(* Value *)
	END_VAR
	VAR_INPUT
		ipContainer	:	ITcVnContainer;	(* Container with TcVnVector4_DINT elements *)
		hrPrev	:	HRESULT;	(* HRESULT indicating the result of previous operations (If SUCCEEDED(hrPrev) equals false, no operation is executed.) *)
	END_VAR

END_FUNCTION

// Functions/Algebraic Container Operations/F_VN_AddToContainerElements/F_VN_AddToContainerElements_TcVnVector4_INT

	{attribute 'TcIecLibraryType'}
	{attribute 'external_name' := 'F_VN_AddToContainerElements_TcVnVector4_INT_GUID_38235CA8_773A_D413_9B6D_513625B9F63E'}
	(* Add a value to each container element. *)
	FUNCTION F_VN_AddToContainerElements_TcVnVector4_INT : HRESULT
	VAR_IN_OUT
		aValue	:	TcVnVector4_INT;	(* Value *)
	END_VAR
	VAR_INPUT
		ipContainer	:	ITcVnContainer;	(* Container with TcVnVector4_INT elements *)
		hrPrev	:	HRESULT;	(* HRESULT indicating the result of previous operations (If SUCCEEDED(hrPrev) equals false, no operation is executed.) *)
	END_VAR

END_FUNCTION

// Functions/Algebraic Container Operations/F_VN_AddToContainerElements/F_VN_AddToContainerElements_TcVnVector4_LREAL

	{attribute 'TcIecLibraryType'}
	{attribute 'external_name' := 'F_VN_AddToContainerElements_TcVnVector4_LREAL_GUID_59A55910_55DA_D0CF_A1CD_BDF48B14B106'}
	(* Add a value to each container element. *)
	FUNCTION F_VN_AddToContainerElements_TcVnVector4_LREAL : HRESULT
	VAR_IN_OUT
		aValue	:	TcVnVector4_LREAL;	(* Value *)
	END_VAR
	VAR_INPUT
		ipContainer	:	ITcVnContainer;	(* Container with TcVnVector4_LREAL elements *)
		hrPrev	:	HRESULT;	(* HRESULT indicating the result of previous operations (If SUCCEEDED(hrPrev) equals false, no operation is executed.) *)
	END_VAR

END_FUNCTION

// Functions/Algebraic Container Operations/F_VN_AddToContainerElements/F_VN_AddToContainerElements_TcVnVector4_REAL

	{attribute 'TcIecLibraryType'}
	{attribute 'external_name' := 'F_VN_AddToContainerElements_TcVnVector4_REAL_GUID_14953B4E_0F43_DB32_96AA_7BFDE4BA2A13'}
	(* Add a value to each container element. *)
	FUNCTION F_VN_AddToContainerElements_TcVnVector4_REAL : HRESULT
	VAR_IN_OUT
		aValue	:	TcVnVector4_REAL;	(* Value *)
	END_VAR
	VAR_INPUT
		ipContainer	:	ITcVnContainer;	(* Container with TcVnVector4_REAL elements *)
		hrPrev	:	HRESULT;	(* HRESULT indicating the result of previous operations (If SUCCEEDED(hrPrev) equals false, no operation is executed.) *)
	END_VAR

END_FUNCTION

// Functions/Algebraic Container Operations/F_VN_AddToContainerElements/F_VN_AddToContainerElements_TcVnVector4_SINT

	{attribute 'TcIecLibraryType'}
	{attribute 'external_name' := 'F_VN_AddToContainerElements_TcVnVector4_SINT_GUID_77808947_A1DF_DA5F_A627_45A690CA9EB2'}
	(* Add a value to each container element. *)
	FUNCTION F_VN_AddToContainerElements_TcVnVector4_SINT : HRESULT
	VAR_IN_OUT
		aValue	:	TcVnVector4_SINT;	(* Value *)
	END_VAR
	VAR_INPUT
		ipContainer	:	ITcVnContainer;	(* Container with TcVnVector4_SINT elements *)
		hrPrev	:	HRESULT;	(* HRESULT indicating the result of previous operations (If SUCCEEDED(hrPrev) equals false, no operation is executed.) *)
	END_VAR

END_FUNCTION

// Functions/Algebraic Container Operations/F_VN_AddToContainerElements/F_VN_AddToContainerElements_TcVnVector4_UINT

	{attribute 'TcIecLibraryType'}
	{attribute 'external_name' := 'F_VN_AddToContainerElements_TcVnVector4_UINT_GUID_3E279758_B798_DA56_AC44_2205B27D4ED9'}
	(* Add a value to each container element. *)
	FUNCTION F_VN_AddToContainerElements_TcVnVector4_UINT : HRESULT
	VAR_IN_OUT
		aValue	:	TcVnVector4_UINT;	(* Value *)
	END_VAR
	VAR_INPUT
		ipContainer	:	ITcVnContainer;	(* Container with TcVnVector4_UINT elements *)
		hrPrev	:	HRESULT;	(* HRESULT indicating the result of previous operations (If SUCCEEDED(hrPrev) equals false, no operation is executed.) *)
	END_VAR

END_FUNCTION

// Functions/Algebraic Container Operations/F_VN_AddToContainerElements/F_VN_AddToContainerElements_TcVnVector4_USINT

	{attribute 'TcIecLibraryType'}
	{attribute 'external_name' := 'F_VN_AddToContainerElements_TcVnVector4_USINT_GUID_18F8356D_1D7E_D3E4_984A_A622A486D99E'}
	(* Add a value to each container element. *)
	FUNCTION F_VN_AddToContainerElements_TcVnVector4_USINT : HRESULT
	VAR_IN_OUT
		aValue	:	TcVnVector4_USINT;	(* Value *)
	END_VAR
	VAR_INPUT
		ipContainer	:	ITcVnContainer;	(* Container with TcVnVector4_USINT elements *)
		hrPrev	:	HRESULT;	(* HRESULT indicating the result of previous operations (If SUCCEEDED(hrPrev) equals false, no operation is executed.) *)
	END_VAR

END_FUNCTION

// Functions/Algebraic Container Operations/F_VN_AddToContainerElements/F_VN_AddToContainerElements_UDINT

	{attribute 'TcIecLibraryType'}
	{attribute 'external_name' := 'F_VN_AddToContainerElements_UDINT_GUID_316D6A2D_D3A9_D9AD_B611_FF08820D03CD'}
	(* Add a value to each container element. *)
	FUNCTION F_VN_AddToContainerElements_UDINT : HRESULT
	VAR_INPUT
		nValue	:	UDINT;	(* Value *)
		ipContainer	:	ITcVnContainer;	(* Container with UDINT elements *)
		hrPrev	:	HRESULT;	(* HRESULT indicating the result of previous operations (If SUCCEEDED(hrPrev) equals false, no operation is executed.) *)
	END_VAR

END_FUNCTION

// Functions/Algebraic Container Operations/F_VN_AddToContainerElements/F_VN_AddToContainerElements_UINT

	{attribute 'TcIecLibraryType'}
	{attribute 'external_name' := 'F_VN_AddToContainerElements_UINT_GUID_C569F72E_F9D4_DC91_8530_B007F80F8B11'}
	(* Add a value to each container element. *)
	FUNCTION F_VN_AddToContainerElements_UINT : HRESULT
	VAR_INPUT
		nValue	:	UINT;	(* Value *)
		ipContainer	:	ITcVnContainer;	(* Container with UINT elements *)
		hrPrev	:	HRESULT;	(* HRESULT indicating the result of previous operations (If SUCCEEDED(hrPrev) equals false, no operation is executed.) *)
	END_VAR

END_FUNCTION

// Functions/Algebraic Container Operations/F_VN_AddToContainerElements/F_VN_AddToContainerElements_ULINT

	{attribute 'TcIecLibraryType'}
	{attribute 'external_name' := 'F_VN_AddToContainerElements_ULINT_GUID_EA1FD331_4923_D56D_B5B0_97F98F96136C'}
	(* Add a value to each container element. *)
	FUNCTION F_VN_AddToContainerElements_ULINT : HRESULT
	VAR_INPUT
		nValue	:	ULINT;	(* Value *)
		ipContainer	:	ITcVnContainer;	(* Container with ULINT elements *)
		hrPrev	:	HRESULT;	(* HRESULT indicating the result of previous operations (If SUCCEEDED(hrPrev) equals false, no operation is executed.) *)
	END_VAR

END_FUNCTION

// Functions/Algebraic Container Operations/F_VN_AddToContainerElements/F_VN_AddToContainerElements_USINT

	{attribute 'TcIecLibraryType'}
	{attribute 'external_name' := 'F_VN_AddToContainerElements_USINT_GUID_3453D20F_2659_DB9B_9F10_DC7E3BA46A8B'}
	(* Add a value to each container element. *)
	FUNCTION F_VN_AddToContainerElements_USINT : HRESULT
	VAR_INPUT
		nValue	:	USINT;	(* Value *)
		ipContainer	:	ITcVnContainer;	(* Container with USINT elements *)
		hrPrev	:	HRESULT;	(* HRESULT indicating the result of previous operations (If SUCCEEDED(hrPrev) equals false, no operation is executed.) *)
	END_VAR

END_FUNCTION

// Functions/Image Analysis/Object Detection/F_VN_AdjustActiveContour

	{attribute 'TcIecLibraryType'}
	{attribute 'external_name' := 'F_VN_AdjustActiveContour_GUID_87080361_5189_D3D0_9045_34EDAC7C1DB1'}
	(* Adjust active contour (snake) in order to minimize its cummulative (internal and external) energy. *)
	FUNCTION F_VN_AdjustActiveContour : HRESULT
	VAR_INPUT
		ipImage	:	ITcVnImage;	(* Source image (1 channel, USINT elements) *)
		ipActiveContour	:	ITcVnContainer;	(* Initial contour, which will be adjusted *)
		fAlpha	:	REAL;	(* Continuity energy coefficient *)
		fBeta	:	REAL;	(* Curvature energy coefficient *)
		fGamma	:	REAL;	(* Image energy coefficient *)
		nWindowWidth	:	UDINT;	(* Window width (3, 5, 7, ...) *)
		nWindowHeight	:	UDINT;	(* Window height (3, 5, 7, ...) *)
		nMaxIterations	:	UDINT;	(* Maximum iterations *)
		bUseGradient	:	BOOL;	(* If true, the gradient magnitude is used as image energy (otherwise: pixel intensity) *)
		hrPrev	:	HRESULT;	(* HRESULT indicating the result of previous operations (If SUCCEEDED(hrPrev) equals false, no operation is executed.) *)
	END_VAR

END_FUNCTION

// Functions/Image Analysis/Object Detection/F_VN_DetectBlobs

	{attribute 'TcIecLibraryType'}
	{attribute 'external_name' := 'F_VN_DetectBlobs_GUID_B6CBB486_3BFA_D359_AD47_E25F509374D8'}
	(* Detects blob-contours. Applies a threshold, a contour search and offers several options for filtering the found contours. Provides easy setup for multiple thresholds and combination of results. *)
	FUNCTION F_VN_DetectBlobs : HRESULT
	VAR_INPUT
		ipSrcImage	:	ITcVnImage;	(* Source image (USINT or REAL, 1 channel or 3 channel (3 channel input is expected to be RGB and internally converted to Gray)) *)
		ipBlobContours	:	REFERENCE TO ITcVnContainer;	(* Returns a container which is filled with the found contours (ContainerType_Vector_Vector_TcVnPoint2_DINT; The elements of this container are single contours. Non-zero interface pointers are reused.) *)
	END_VAR
	VAR_IN_OUT
		stParams	:	TcVnParamsBlobDetection;	(* Parameters to filter the detected contours. *)
	END_VAR
	VAR_INPUT
		hrPrev	:	HRESULT;	(* HRESULT indicating the result of previous operations (If SUCCEEDED(hrPrev) equals false, no operation is executed.) *)
	END_VAR

END_FUNCTION

// Functions/Image Analysis/Object Detection/F_VN_DetectBlobsExp

	{attribute 'TcIecLibraryType'}
	{attribute 'external_name' := 'F_VN_DetectBlobsExp_GUID_93B114AF_ED91_D3C9_87F0_32F15F980672'}
	(* Detects blob-contours. Applies a threshold, a contour search and offers several options for filtering the found contours. Provides easy setup for multiple thresholds and combination of results. (expert function) *)
	FUNCTION F_VN_DetectBlobsExp : HRESULT
	VAR_INPUT
		ipSrcImage	:	ITcVnImage;	(* Source image (USINT or REAL, 1 channel or 3 channel (3 channel input is expected to be RGB and internally converted to Gray)) *)
		ipBlobContours	:	REFERENCE TO ITcVnContainer;	(* Returns a container which is filled with the found contours (ContainerType_Vector_Vector_TcVnPoint2_DINT; The elements of this container are single contours. Non-zero interface pointers are reused.) *)
	END_VAR
	VAR_IN_OUT
		stParams	:	TcVnParamsBlobDetection;	(* Parameters to filter the detected contours. *)
		aOffset	:	TcVnPoint;	(* Offset by which every contour point is shifted *)
	END_VAR
	VAR_INPUT
		hrPrev	:	HRESULT;	(* HRESULT indicating the result of previous operations (If SUCCEEDED(hrPrev) equals false, no operation is executed.) *)
	END_VAR

END_FUNCTION

// Functions/Image Analysis/Object Detection/F_VN_FindContourHierarchyExp

	{attribute 'TcIecLibraryType'}
	{attribute 'external_name' := 'F_VN_FindContourHierarchyExp_GUID_FBD38625_FC4B_D014_827E_A5077045F0F0'}
	(* Search for object contours in a binary image and determine their hierarchical relationship. (expert function) *)
	FUNCTION F_VN_FindContourHierarchyExp : HRESULT
	VAR_INPUT
		ipSrcImage	:	ITcVnImage;	(* Source image (1 channel, binary) *)
		ipContours	:	REFERENCE TO ITcVnContainer;	(* Returns a container which is filled with the found contours (ContainerType_Vector_Vector_TcVnPoint2_DINT; The elements of this container are single contours. Non-zero interface pointers are reused.) *)
		ipHierarchy	:	REFERENCE TO ITcVnContainer;	(* Returns a container which is filled with information on the found contours' hierarchy (ContainerType_Vector_TcVnVector4_DINT; The elements of this container are four-dimensional vectors containing the 0-based indices of the next [0] and the previous contour [1] at the same level, the first child [2], and the parent [3]. Non-zero interface pointers are reused.) *)
		eRetrievalMode	:	ETcVnContourRetrievalMode;	(* Specifies which contours are retrieved and how their relationship is encoded *)
		eApproximationMethod	:	ETcVnContourApproximationMethod;	(* Contour encoding *)
	END_VAR
	VAR_IN_OUT
		aOffset	:	TcVnPoint;	(* Offset by which every contour point is shifted *)
	END_VAR
	VAR_INPUT
		hrPrev	:	HRESULT;	(* HRESULT indicating the result of previous operations (If SUCCEEDED(hrPrev) equals false, no operation is executed.) *)
	END_VAR

END_FUNCTION

// Functions/Image Analysis/Object Detection/F_VN_FindContours

	{attribute 'TcIecLibraryType'}
	{attribute 'external_name' := 'F_VN_FindContours_GUID_9318AB52_4BB7_D327_B4E5_0D4368BA0A03'}
	(* Search for object contours in a binary image. Returns only external contours. *)
	FUNCTION F_VN_FindContours : HRESULT
	VAR_INPUT
		ipSrcImage	:	ITcVnImage;	(* Source image (1 channel, binary) *)
		ipContours	:	REFERENCE TO ITcVnContainer;	(* Returns a container which is filled with the found contours (ContainerType_Vector_Vector_TcVnPoint2_DINT; The elements of this container are single contours. Non-zero interface pointers are reused.) *)
		hrPrev	:	HRESULT;	(* HRESULT indicating the result of previous operations (If SUCCEEDED(hrPrev) equals false, no operation is executed.) *)
	END_VAR

END_FUNCTION

// Functions/Image Analysis/Object Detection/F_VN_FindContoursExp

	{attribute 'TcIecLibraryType'}
	{attribute 'external_name' := 'F_VN_FindContoursExp_GUID_E31A68CE_20ED_D131_90FE_F3DBE5C5326D'}
	(* Search for object contours in a binary image. (expert function) *)
	FUNCTION F_VN_FindContoursExp : HRESULT
	VAR_INPUT
		ipSrcImage	:	ITcVnImage;	(* Source image (1 channel, binary) *)
		ipContours	:	REFERENCE TO ITcVnContainer;	(* Returns a container which is filled with the found contours (ContainerType_Vector_Vector_TcVnPoint2_DINT; The elements of this container are single contours. Non-zero interface pointers are reused.) *)
		eRetrievalMode	:	ETcVnContourRetrievalMode;	(* Specifies which contours are retrieved and how their relationship is encoded *)
		eApproximationMethod	:	ETcVnContourApproximationMethod;	(* Contour encoding *)
	END_VAR
	VAR_IN_OUT
		aOffset	:	TcVnPoint;	(* Offset by which every contour point is shifted *)
	END_VAR
	VAR_INPUT
		hrPrev	:	HRESULT;	(* HRESULT indicating the result of previous operations (If SUCCEEDED(hrPrev) equals false, no operation is executed.) *)
	END_VAR

END_FUNCTION

// Functions/Image Analysis/Object Detection/F_VN_HoughCircles

	{attribute 'TcIecLibraryType'}
	{attribute 'external_name' := 'F_VN_HoughCircles_GUID_A989ED23_5F7C_D23B_A00A_F7431317F8BD'}
	(* Search for circles using the Hough transform. *)
	FUNCTION F_VN_HoughCircles : HRESULT
	VAR_INPUT
		ipSrcImage	:	ITcVnImage;	(* Source image (USINT, 1 channel, gray-level) *)
		ipCircles	:	REFERENCE TO ITcVnContainer;	(* Returns a container which is filled with the found circles (ContainerType_Vector_TcVnVector3_REAL; Each container element contains the x coordinate of the circle center [0], the y coordinate of the circle center [1], and the radius [2], respectively. Non-zero interface pointers are reused.) *)
		fInvAccuRatio	:	LREAL;	(* Inverted ratio of the accumulator size in relation to the source image's size (must be > 0. A value of 2 means that the size is halved in both directions.) *)
		fMinDist	:	LREAL;	(* Smallest allowed distance of two circles (must be > 0) *)
		hrPrev	:	HRESULT;	(* HRESULT indicating the result of previous operations (If SUCCEEDED(hrPrev) equals false, no operation is executed.) *)
	END_VAR

END_FUNCTION

// Functions/Image Analysis/Object Detection/F_VN_HoughCirclesExp

	{attribute 'TcIecLibraryType'}
	{attribute 'external_name' := 'F_VN_HoughCirclesExp_GUID_9EA58FE1_B06A_D9D9_BFBA_26541DE4A688'}
	(* Search for circles using the Hough transform. (expert function) *)
	FUNCTION F_VN_HoughCirclesExp : HRESULT
	VAR_INPUT
		ipSrcImage	:	ITcVnImage;	(* Source image (USINT, 1 channel, gray-level) *)
		ipCircles	:	REFERENCE TO ITcVnContainer;	(* Returns a container which is filled with the found circles (ContainerType_Vector_TcVnVector3_REAL; Each container element contains the x coordinate of the circle center [0], the y coordinate of the circle center [1], and the radius [2], respectively. Non-zero interface pointers are reused.) *)
		fInvAccuRatio	:	LREAL;	(* Inverted ratio of the accumulator size in relation to the source image's size (must be > 0. A value of 2 means that the size is halved in both directions.) *)
		fMinDist	:	LREAL;	(* Smallest allowed distance of two circles (must be > 0) *)
		eHoughMethod	:	ETcVnHoughMethod;	(* Hough method to use (GRADIENT or GRADIENT_ALT) *)
		fParam1	:	LREAL;	(* First method specific parameter (GRADIENT, GRADIENT_ALT: upper threshold for canny edge detection, which must be > 0) *)
		fParam2	:	LREAL;	(* Second method specific parameter (GRADIENT: accumulator threshold for detecting circle centers, which must be > 0. GRADIENT_ALT: required circle perfectness, which must be > 0 and < 1, 1 would be a perfect circle) *)
		nMinRadius	:	UDINT;	(* Minimum circle radius allowed *)
		nMaxRadius	:	UDINT;	(* Maximum circle radius allowed (if 0, the value is internally set to max(image rows, image columns)) *)
		hrPrev	:	HRESULT;	(* HRESULT indicating the result of previous operations (If SUCCEEDED(hrPrev) equals false, no operation is executed.) *)
	END_VAR

END_FUNCTION

// Functions/Image Analysis/Object Detection/F_VN_HoughLines

	{attribute 'TcIecLibraryType'}
	{attribute 'external_name' := 'F_VN_HoughLines_GUID_19380114_BB0F_DEE7_BACB_A274896AD30D'}
	(* Search for lines using the standard Hough transform. *)
	FUNCTION F_VN_HoughLines : HRESULT
	VAR_INPUT
		ipSrcImage	:	ITcVnImage;	(* Source image (USINT, 1 channel, binary, may be modified by the function) *)
		ipLines	:	REFERENCE TO ITcVnContainer;	(* Returns a container which is filled with the found lines (ContainerType_Vector_TcVnVector2_REAL; Each container element contains the distance from the origin [0] in pixels and the rotation angle [1] in radians, respectively. Non-zero interface pointers are reused.) *)
		fDistRes	:	LREAL;	(* Distance resolution of the accumulator (in pixels, must be > 0) *)
		fAngleRes	:	LREAL;	(* Angle resolution of the accumulator (in radians, must be > 0) *)
		nAccuThreshold	:	UDINT;	(* Accumulator threshold *)
		hrPrev	:	HRESULT;	(* HRESULT indicating the result of previous operations (If SUCCEEDED(hrPrev) equals false, no operation is executed.) *)
	END_VAR

END_FUNCTION

// Functions/Image Analysis/Object Detection/F_VN_HoughLinesExp

	{attribute 'TcIecLibraryType'}
	{attribute 'external_name' := 'F_VN_HoughLinesExp_GUID_33E62D5A_29F7_DF75_A7A0_60B6FB7AF93D'}
	(* Search for lines using the standard Hough transform. (expert function) *)
	FUNCTION F_VN_HoughLinesExp : HRESULT
	VAR_INPUT
		ipSrcImage	:	ITcVnImage;	(* Source image (USINT, 1 channel, binary, may be modified by the function) *)
		ipLines	:	REFERENCE TO ITcVnContainer;	(* Returns a container which is filled with the found lines (ContainerType_Vector_TcVnVector2_REAL; Each container element contains the distance from the origin [0] in pixels and the rotation angle [1] in radians, respectively. Non-zero interface pointers are reused.) *)
		fDistRes	:	LREAL;	(* Distance resolution of the accumulator (in pixels, must be > 0) *)
		fAngleRes	:	LREAL;	(* Angle resolution of the accumulator (in radians, must be > 0) *)
		nAccuThreshold	:	UDINT;	(* Accumulator threshold *)
		fDistResDiv	:	LREAL;	(* Divisor of the distance resolution for the multi-scale Hough transform (>= 0, must be > 0 if fAngleResDiv is > 0) *)
		fAngleResDiv	:	LREAL;	(* Divisor of the angle resolution for the multi-scale Hough transform (>= 0, must be > 0 if fDistResDiv is > 0) *)
		hrPrev	:	HRESULT;	(* HRESULT indicating the result of previous operations (If SUCCEEDED(hrPrev) equals false, no operation is executed.) *)
	END_VAR

END_FUNCTION

// Functions/Image Analysis/Object Detection/F_VN_HoughLinesP

	{attribute 'TcIecLibraryType'}
	{attribute 'external_name' := 'F_VN_HoughLinesP_GUID_CD259D33_7801_D5D3_8468_EEBA188ECF94'}
	(* Search for line segments using the probabilistic Hough transform. *)
	FUNCTION F_VN_HoughLinesP : HRESULT
	VAR_INPUT
		ipSrcImage	:	ITcVnImage;	(* Source image (USINT, 1 channel, binary, may be modified by the function) *)
		ipLines	:	REFERENCE TO ITcVnContainer;	(* Returns a container which is filled with the found line segments (ContainerType_Vector_TcVnVector4_DINT; Each container element contains the two ending points. Non-zero interface pointers are reused.) *)
		fDistRes	:	LREAL;	(* Distance resolution of the accumulator (in pixels, must be > 0) *)
		fAngleRes	:	LREAL;	(* Angle resolution of the accumulator (in radians, must be > 0) *)
		nAccuThreshold	:	UDINT;	(* Accumulator threshold *)
		hrPrev	:	HRESULT;	(* HRESULT indicating the result of previous operations (If SUCCEEDED(hrPrev) equals false, no operation is executed.) *)
	END_VAR

END_FUNCTION

// Functions/Image Analysis/Object Detection/F_VN_HoughLinesPExp

	{attribute 'TcIecLibraryType'}
	{attribute 'external_name' := 'F_VN_HoughLinesPExp_GUID_404CFB76_923E_D49E_A094_13154A22EBA6'}
	(* Search for line segments using the probabilistic Hough transform. (expert function) *)
	FUNCTION F_VN_HoughLinesPExp : HRESULT
	VAR_INPUT
		ipSrcImage	:	ITcVnImage;	(* Source image (USINT, 1 channel, binary, may be modified by the function) *)
		ipLines	:	REFERENCE TO ITcVnContainer;	(* Returns a container which is filled with the found line segments (ContainerType_Vector_TcVnVector4_DINT; Each container element contains the two ending points. Non-zero interface pointers are reused.) *)
		fDistRes	:	LREAL;	(* Distance resolution of the accumulator (in pixels, must be > 0) *)
		fAngleRes	:	LREAL;	(* Angle resolution of the accumulator (in radians, must be > 0) *)
		nAccuThreshold	:	UDINT;	(* Accumulator threshold *)
		fMinLineLength	:	LREAL;	(* Minimum line length to search for *)
		fMaxLineGap	:	LREAL;	(* Maximum gap between points on the same line *)
		hrPrev	:	HRESULT;	(* HRESULT indicating the result of previous operations (If SUCCEEDED(hrPrev) equals false, no operation is executed.) *)
	END_VAR

END_FUNCTION

// Functions/Image Analysis/Object Detection/F_VN_MatchImageHuMoments

	{attribute 'TcIecLibraryType'}
	{attribute 'external_name' := 'F_VN_MatchImageHuMoments_GUID_FE0D37C9_15D4_D533_A9A6_FFE07C999981'}
	(* Compare two images using the Hu moment invariants. *)
	FUNCTION F_VN_MatchImageHuMoments : HRESULT
	VAR_INPUT
		ipImage1	:	ITcVnImage;	(* First image (1 channel) *)
		ipImage2	:	ITcVnImage;	(* Second image (1 channel) *)
		eComparisonMethod	:	ETcVnContoursMatchComparisonMethod;	(* Method used for comparing the Hu moment invariants of the images *)
	END_VAR
	VAR_IN_OUT
		fDissimilarity	:	LREAL;	(* Returns the dissimilarity of the image Hu moment invariants depending on the chosen comparison method *)
	END_VAR
	VAR_INPUT
		hrPrev	:	HRESULT;	(* HRESULT indicating the result of previous operations (If SUCCEEDED(hrPrev) equals false, no operation is executed.) *)
	END_VAR

END_FUNCTION

// Functions/Image Analysis/Object Detection/F_VN_MatchTemplate

	{attribute 'TcIecLibraryType'}
	{attribute 'external_name' := 'F_VN_MatchTemplate_GUID_5B62EF07_B480_D00E_A874_5DC920C704CE'}
	(* Match a template image with every location in the source image (using the TCVN_TMM_CCORR_NORMED method) and save the comparison results. *)
	FUNCTION F_VN_MatchTemplate : HRESULT
	VAR_INPUT
		ipSrcImage	:	ITcVnImage;	(* Source image (USINT or REAL, 1 or 3 channels) *)
		ipTemplateImage	:	ITcVnImage;	(* Template image (same type as ipSrcImage, smaller width and height) *)
		ipResultImage	:	REFERENCE TO ITcVnImage;	(* Returns the result image (REAL, normalized to [0..1], 1 channel, dimensions: (ipSrcImage.width - ipTemplateImage.width + 1) x (ipSrcImage.height - ipTemplateImage.height + 1). The best match is the global maximum. The position in ipResultImage is the top-left corner of ipTemplateImage position in ipSrcImage) *)
		hrPrev	:	HRESULT;	(* HRESULT indicating the result of previous operations (If SUCCEEDED(hrPrev) equals false, no operation is executed.) *)
	END_VAR

END_FUNCTION

// Functions/Image Analysis/Object Detection/F_VN_MatchTemplateExp

	{attribute 'TcIecLibraryType'}
	{attribute 'external_name' := 'F_VN_MatchTemplateExp_GUID_AD09D891_9A55_D2B3_9383_DC2062AF9171'}
	(* Match a template image with every location in the source image and save the comparison results. (expert function) *)
	FUNCTION F_VN_MatchTemplateExp : HRESULT
	VAR_INPUT
		ipSrcImage	:	ITcVnImage;	(* Source image (USINT or REAL, 1 or 3 channels) *)
		ipTemplateImage	:	ITcVnImage;	(* Template image (same type as ipSrcImage, smaller width and height) *)
		ipResultImage	:	REFERENCE TO ITcVnImage;	(* Returns the result image (REAL, 1 channel, dimensions: (ipSrcImage.width - ipTemplateImage.width + 1) x (ipSrcImage.height - ipTemplateImage.height + 1). The best match is the global minimum (SQDIFF(_NORMED)) or maximum (CCORR(_NORMED), CCOEFF(_NORMED)). The position in ipResultImage is the top-left corner of ipTemplateImage position in ipSrcImage) *)
		eMatchMethod	:	ETcVnTemplateMatchMethod;	(* Specifies the template match method *)
		ipTemplateMask	:	ITcVnImage;	(* Optional mask for ipTemplateImage (same type and size as ipTemplateImage) *)
		hrPrev	:	HRESULT;	(* HRESULT indicating the result of previous operations (If SUCCEEDED(hrPrev) equals false, no operation is executed.) *)
	END_VAR

END_FUNCTION

// Functions/Image Analysis/Object Detection/F_VN_MatchTemplateAndEvaluate

	{attribute 'TcIecLibraryType'}
	{attribute 'external_name' := 'F_VN_MatchTemplateAndEvaluate_GUID_4F1F6206_B887_D211_A921_D9457AB3815E'}
	(* Match a template image with every location in the source image (using the TCVN_TMM_CCORR_NORMED method) and evaluate the comparison results. Returns a sorted list of possible matches (best match first). *)
	FUNCTION F_VN_MatchTemplateAndEvaluate : HRESULT
	VAR_INPUT
		ipSrcImage	:	ITcVnImage;	(* Source image (USINT or REAL, 1 or 3 channels) *)
		ipTemplateImage	:	ITcVnImage;	(* Template image (same type as ipSrcImage, smaller width and height) *)
		ipMatches	:	REFERENCE TO ITcVnContainer;	(* Returns the matching positions (ContainerType_Vector_TcVnPoint2_DINT, where each element represents the top-left corner of ipTemplateImage) in ipSrcImage, sorted by relevance (best match first) *)
		fMatchThreshold	:	REAL;	(* Threshold to separate relevant from irrelevant matches (0..1, 1.0  would be a perfect match. To find a suitable value, you could evaluate some sample result images of F_VN_MatchTemplate.) *)
		hrPrev	:	HRESULT;	(* HRESULT indicating the result of previous operations (If SUCCEEDED(hrPrev) equals false, no operation is executed.) *)
	END_VAR

END_FUNCTION

// Functions/Image Analysis/Object Detection/F_VN_MatchTemplateAndEvaluateExp

	{attribute 'TcIecLibraryType'}
	{attribute 'external_name' := 'F_VN_MatchTemplateAndEvaluateExp_GUID_C9F60D55_13B5_D04B_91EA_4287EADC2DEF'}
	(* Match a template image with every location in the source image and evaluate the comparison results. Returns a sorted list of possible matches (best match first). (expert function) *)
	FUNCTION F_VN_MatchTemplateAndEvaluateExp : HRESULT
	VAR_INPUT
		ipSrcImage	:	ITcVnImage;	(* Source image (USINT or REAL, 1 or 3 channels) *)
		ipTemplateImage	:	ITcVnImage;	(* Template image (same type as ipSrcImage, smaller width and height) *)
		ipMatches	:	REFERENCE TO ITcVnContainer;	(* Returns the matching positions (ContainerType_Vector_TcVnPoint2_DINT, where each element represents the top-left corner of ipTemplateImage) in ipSrcImage, sorted by relevance (best match first) *)
		fMatchThreshold	:	REAL;	(* Threshold to separate relevant from irrelevant matches (0..1 for NORMED methods, otherwise dependent on template size and content. To find a suitable value, you could evaluate some sample result images of F_VN_MatchTemplateExp.) *)
		eMatchMethod	:	ETcVnTemplateMatchMethod;	(* Specifies the template match method *)
		ipTemplateMask	:	ITcVnImage;	(* Optional mask for ipTemplateImage (same type and size as ipTemplateImage) *)
		fScaleFactor	:	REAL;	(* Factor (0..1] to reduce source and template image width and height for better performance (but less accuracy!) *)
		eInterpolationType	:	ETcVnInterpolationType;	(* Image resize interpolation type (only used if fScaleFactor != 1, TCVN_IT_BILINEAR recommended for most cases) *)
		ipMatchValues	:	REFERENCE TO ITcVnContainer;	(* Optionally returns the matching values (ContainerType_Vector_REAL, same size and sort order as ipMatches. Set to 0 if not required.) *)
		hrPrev	:	HRESULT;	(* HRESULT indicating the result of previous operations (If SUCCEEDED(hrPrev) equals false, no operation is executed.) *)
	END_VAR

END_FUNCTION

// Functions/Basic Container Operations/F_VN_AppendToContainer/F_VN_AppendToContainer_ITcVnContainer

	{attribute 'TcIecLibraryType'}
	{attribute 'external_name' := 'F_VN_AppendToContainer_ITcVnContainer_GUID_93F08F23_37DF_D41B_B8C5_037FAC5A848C'}
	(* Append a single element to a container or concatenate containers (if ipElement has the same typeId as ipContainer). *)
	FUNCTION F_VN_AppendToContainer_ITcVnContainer : HRESULT
	VAR_INPUT
		ipElement	:	ITcVnContainer;	(* Single element to append to ipContainer or container with several elements to be concatenated *)
		ipContainer	:	ITcVnContainer;	(* Container to which the element(s) will be appended *)
		hrPrev	:	HRESULT;	(* HRESULT indicating the result of previous operations (If SUCCEEDED(hrPrev) equals false, no operation is executed.) *)
	END_VAR

END_FUNCTION

// Functions/Basic Container Operations/F_VN_AppendToContainer/F_VN_AppendToContainer_ITcVnForwardIterator

	{attribute 'TcIecLibraryType'}
	{attribute 'external_name' := 'F_VN_AppendToContainer_ITcVnForwardIterator_GUID_F37F6501_ABBB_D6BB_909B_7622AC495989'}
	(* Append a single element (represented by an iterator)to a container. *)
	FUNCTION F_VN_AppendToContainer_ITcVnForwardIterator : HRESULT
	VAR_INPUT
		ipElement	:	ITcVnForwardIterator;	(* Single element to append to ipContainer *)
		ipContainer	:	ITcVnContainer;	(* Container to which the element(s) will be appended *)
		hrPrev	:	HRESULT;	(* HRESULT indicating the result of previous operations (If SUCCEEDED(hrPrev) equals false, no operation is executed.) *)
	END_VAR

END_FUNCTION

// Functions/Basic Container Operations/F_VN_AppendToContainer/F_VN_AppendToContainer_DINT

	{attribute 'TcIecLibraryType'}
	{attribute 'external_name' := 'F_VN_AppendToContainer_DINT_GUID_5E62B518_4D4D_D6B6_8949_8B38FC59108F'}
	(* Append a single element of type DINT to a container. *)
	FUNCTION F_VN_AppendToContainer_DINT : HRESULT
	VAR_INPUT
		nElement	:	DINT;	(* Single element to append to ipContainer *)
		ipContainer	:	ITcVnContainer;	(* Container to which the element will be appended *)
		hrPrev	:	HRESULT;	(* HRESULT indicating the result of previous operations (If SUCCEEDED(hrPrev) equals false, no operation is executed.) *)
	END_VAR

END_FUNCTION

// Functions/Basic Container Operations/F_VN_AppendToContainer/F_VN_AppendToContainer_INT

	{attribute 'TcIecLibraryType'}
	{attribute 'external_name' := 'F_VN_AppendToContainer_INT_GUID_84232AEA_29C0_D7D4_94FF_A7197598429A'}
	(* Append a single element of type INT to a container. *)
	FUNCTION F_VN_AppendToContainer_INT : HRESULT
	VAR_INPUT
		nElement	:	INT;	(* Single element to append to ipContainer *)
		ipContainer	:	ITcVnContainer;	(* Container to which the element will be appended *)
		hrPrev	:	HRESULT;	(* HRESULT indicating the result of previous operations (If SUCCEEDED(hrPrev) equals false, no operation is executed.) *)
	END_VAR

END_FUNCTION

// Functions/Basic Container Operations/F_VN_AppendToContainer/F_VN_AppendToContainer_ITcVnImage

	{attribute 'TcIecLibraryType'}
	{attribute 'external_name' := 'F_VN_AppendToContainer_ITcVnImage_GUID_02CBB15B_5F5A_D0CB_A558_01318AB069E6'}
	(* Append a single element of type ITcVnImage to a container. *)
	FUNCTION F_VN_AppendToContainer_ITcVnImage : HRESULT
	VAR_INPUT
		ipElement	:	ITcVnImage;	(* Single element to append to ipContainer *)
		ipContainer	:	ITcVnContainer;	(* Container to which the element will be appended *)
		hrPrev	:	HRESULT;	(* HRESULT indicating the result of previous operations (If SUCCEEDED(hrPrev) equals false, no operation is executed.) *)
	END_VAR

END_FUNCTION

// Functions/Basic Container Operations/F_VN_AppendToContainer/F_VN_AppendToContainer_LREAL

	{attribute 'TcIecLibraryType'}
	{attribute 'external_name' := 'F_VN_AppendToContainer_LREAL_GUID_A9AFAB30_EE50_DA6E_BCC8_0E01ECC80DB5'}
	(* Append a single element of type LREAL to a container. *)
	FUNCTION F_VN_AppendToContainer_LREAL : HRESULT
	VAR_INPUT
		fElement	:	LREAL;	(* Single element to append to ipContainer *)
		ipContainer	:	ITcVnContainer;	(* Container to which the element will be appended *)
		hrPrev	:	HRESULT;	(* HRESULT indicating the result of previous operations (If SUCCEEDED(hrPrev) equals false, no operation is executed.) *)
	END_VAR

END_FUNCTION

// Functions/Basic Container Operations/F_VN_AppendToContainer/F_VN_AppendToContainer_REAL

	{attribute 'TcIecLibraryType'}
	{attribute 'external_name' := 'F_VN_AppendToContainer_REAL_GUID_B0AA736F_A597_DC9A_A54C_CB918F86921F'}
	(* Append a single element of type REAL to a container. *)
	FUNCTION F_VN_AppendToContainer_REAL : HRESULT
	VAR_INPUT
		fElement	:	REAL;	(* Single element to append to ipContainer *)
		ipContainer	:	ITcVnContainer;	(* Container to which the element will be appended *)
		hrPrev	:	HRESULT;	(* HRESULT indicating the result of previous operations (If SUCCEEDED(hrPrev) equals false, no operation is executed.) *)
	END_VAR

END_FUNCTION

// Functions/Basic Container Operations/F_VN_AppendToContainer/F_VN_AppendToContainer_SINT

	{attribute 'TcIecLibraryType'}
	{attribute 'external_name' := 'F_VN_AppendToContainer_SINT_GUID_368FE265_171C_D030_A1AB_A648313D276D'}
	(* Append a single element of type SINT to a container. *)
	FUNCTION F_VN_AppendToContainer_SINT : HRESULT
	VAR_INPUT
		nElement	:	SINT;	(* Single element to append to ipContainer *)
		ipContainer	:	ITcVnContainer;	(* Container to which the element will be appended *)
		hrPrev	:	HRESULT;	(* HRESULT indicating the result of previous operations (If SUCCEEDED(hrPrev) equals false, no operation is executed.) *)
	END_VAR

END_FUNCTION

// Functions/Basic Container Operations/F_VN_AppendToContainer/F_VN_AppendToContainer_TcVnDMatch

	{attribute 'TcIecLibraryType'}
	{attribute 'external_name' := 'F_VN_AppendToContainer_TcVnDMatch_GUID_2C89D61A_534B_D7BF_ACF8_24206D187F93'}
	(* Append a single element of type TcVnDMatch to a container. *)
	FUNCTION F_VN_AppendToContainer_TcVnDMatch : HRESULT
	VAR_IN_OUT
		stElement	:	TcVnDMatch;	(* Single element to append to ipContainer *)
	END_VAR
	VAR_INPUT
		ipContainer	:	ITcVnContainer;	(* Container to which the element will be appended *)
		hrPrev	:	HRESULT;	(* HRESULT indicating the result of previous operations (If SUCCEEDED(hrPrev) equals false, no operation is executed.) *)
	END_VAR

END_FUNCTION

// Functions/Basic Container Operations/F_VN_AppendToContainer/F_VN_AppendToContainer_TcVnKeyPoint

	{attribute 'TcIecLibraryType'}
	{attribute 'external_name' := 'F_VN_AppendToContainer_TcVnKeyPoint_GUID_C511D5FE_7D76_D29C_B96B_9E660CA5CB7F'}
	(* Append a single element of type TcVnKeyPoint to a container. *)
	FUNCTION F_VN_AppendToContainer_TcVnKeyPoint : HRESULT
	VAR_IN_OUT
		stElement	:	TcVnKeyPoint;	(* Single element to append to ipContainer *)
	END_VAR
	VAR_INPUT
		ipContainer	:	ITcVnContainer;	(* Container to which the element will be appended *)
		hrPrev	:	HRESULT;	(* HRESULT indicating the result of previous operations (If SUCCEEDED(hrPrev) equals false, no operation is executed.) *)
	END_VAR

END_FUNCTION

// Functions/Basic Container Operations/F_VN_AppendToContainer/F_VN_AppendToContainer_TcVnPoint2_DINT

	{attribute 'TcIecLibraryType'}
	{attribute 'external_name' := 'F_VN_AppendToContainer_TcVnPoint2_DINT_GUID_FA3B6F66_E9B5_DB0A_8BA4_6B6F23830075'}
	(* Append a single element of type TcVnPoint2_DINT to a container. *)
	FUNCTION F_VN_AppendToContainer_TcVnPoint2_DINT : HRESULT
	VAR_IN_OUT
		aElement	:	TcVnPoint2_DINT;	(* Single element to append to ipContainer *)
	END_VAR
	VAR_INPUT
		ipContainer	:	ITcVnContainer;	(* Container to which the element will be appended *)
		hrPrev	:	HRESULT;	(* HRESULT indicating the result of previous operations (If SUCCEEDED(hrPrev) equals false, no operation is executed.) *)
	END_VAR

END_FUNCTION

// Functions/Basic Container Operations/F_VN_AppendToContainer/F_VN_AppendToContainer_TcVnPoint2_LREAL

	{attribute 'TcIecLibraryType'}
	{attribute 'external_name' := 'F_VN_AppendToContainer_TcVnPoint2_LREAL_GUID_0EF98D40_921B_D2DC_933F_BDD456F72BBE'}
	(* Append a single element of type TcVnPoint2_LREAL to a container. *)
	FUNCTION F_VN_AppendToContainer_TcVnPoint2_LREAL : HRESULT
	VAR_IN_OUT
		aElement	:	TcVnPoint2_LREAL;	(* Single element to append to ipContainer *)
	END_VAR
	VAR_INPUT
		ipContainer	:	ITcVnContainer;	(* Container to which the element will be appended *)
		hrPrev	:	HRESULT;	(* HRESULT indicating the result of previous operations (If SUCCEEDED(hrPrev) equals false, no operation is executed.) *)
	END_VAR

END_FUNCTION

// Functions/Basic Container Operations/F_VN_AppendToContainer/F_VN_AppendToContainer_TcVnPoint2_REAL

	{attribute 'TcIecLibraryType'}
	{attribute 'external_name' := 'F_VN_AppendToContainer_TcVnPoint2_REAL_GUID_B72DEDE2_EE82_D692_B849_1B007AC42BF4'}
	(* Append a single element of type TcVnPoint2_REAL to a container. *)
	FUNCTION F_VN_AppendToContainer_TcVnPoint2_REAL : HRESULT
	VAR_IN_OUT
		aElement	:	TcVnPoint2_REAL;	(* Single element to append to ipContainer *)
	END_VAR
	VAR_INPUT
		ipContainer	:	ITcVnContainer;	(* Container to which the element will be appended *)
		hrPrev	:	HRESULT;	(* HRESULT indicating the result of previous operations (If SUCCEEDED(hrPrev) equals false, no operation is executed.) *)
	END_VAR

END_FUNCTION

// Functions/Basic Container Operations/F_VN_AppendToContainer/F_VN_AppendToContainer_TcVnPoint3_LREAL

	{attribute 'TcIecLibraryType'}
	{attribute 'external_name' := 'F_VN_AppendToContainer_TcVnPoint3_LREAL_GUID_5B8CECF8_1EE3_D5AD_99B1_12A279F782DA'}
	(* Append a single element of type TcVnPoint3_LREAL to a container. *)
	FUNCTION F_VN_AppendToContainer_TcVnPoint3_LREAL : HRESULT
	VAR_IN_OUT
		aElement	:	TcVnPoint3_LREAL;	(* Single element to append to ipContainer *)
	END_VAR
	VAR_INPUT
		ipContainer	:	ITcVnContainer;	(* Container to which the element will be appended *)
		hrPrev	:	HRESULT;	(* HRESULT indicating the result of previous operations (If SUCCEEDED(hrPrev) equals false, no operation is executed.) *)
	END_VAR

END_FUNCTION

// Functions/Basic Container Operations/F_VN_AppendToContainer/F_VN_AppendToContainer_TcVnPoint3_REAL

	{attribute 'TcIecLibraryType'}
	{attribute 'external_name' := 'F_VN_AppendToContainer_TcVnPoint3_REAL_GUID_47547ECC_5ED2_D213_8561_55E302AA01ED'}
	(* Append a single element of type TcVnPoint3_REAL to a container. *)
	FUNCTION F_VN_AppendToContainer_TcVnPoint3_REAL : HRESULT
	VAR_IN_OUT
		aElement	:	TcVnPoint3_REAL;	(* Single element to append to ipContainer *)
	END_VAR
	VAR_INPUT
		ipContainer	:	ITcVnContainer;	(* Container to which the element will be appended *)
		hrPrev	:	HRESULT;	(* HRESULT indicating the result of previous operations (If SUCCEEDED(hrPrev) equals false, no operation is executed.) *)
	END_VAR

END_FUNCTION

// Functions/Basic Container Operations/F_VN_AppendToContainer/F_VN_AppendToContainer_TcVnRectangle_DINT

	{attribute 'TcIecLibraryType'}
	{attribute 'external_name' := 'F_VN_AppendToContainer_TcVnRectangle_DINT_GUID_5F295922_7114_D051_93E1_48FD2A517D4E'}
	(* Append a single element of type TcVnRectangle_DINT to a container. *)
	FUNCTION F_VN_AppendToContainer_TcVnRectangle_DINT : HRESULT
	VAR_IN_OUT
		stElement	:	TcVnRectangle_DINT;	(* Single element to append to ipContainer *)
	END_VAR
	VAR_INPUT
		ipContainer	:	ITcVnContainer;	(* Container to which the element will be appended *)
		hrPrev	:	HRESULT;	(* HRESULT indicating the result of previous operations (If SUCCEEDED(hrPrev) equals false, no operation is executed.) *)
	END_VAR

END_FUNCTION

// Functions/Basic Container Operations/F_VN_AppendToContainer/F_VN_AppendToContainer_TcVnRotatedRectangle

	{attribute 'TcIecLibraryType'}
	{attribute 'external_name' := 'F_VN_AppendToContainer_TcVnRotatedRectangle_GUID_6FEAA642_D911_DCE9_80D8_518699F3F522'}
	(* Append a single element of type TcVnRotatedRectangle to a container. *)
	FUNCTION F_VN_AppendToContainer_TcVnRotatedRectangle : HRESULT
	VAR_IN_OUT
		stElement	:	TcVnRotatedRectangle;	(* Single element to append to ipContainer *)
	END_VAR
	VAR_INPUT
		ipContainer	:	ITcVnContainer;	(* Container to which the element will be appended *)
		hrPrev	:	HRESULT;	(* HRESULT indicating the result of previous operations (If SUCCEEDED(hrPrev) equals false, no operation is executed.) *)
	END_VAR

END_FUNCTION

// Functions/Basic Container Operations/F_VN_AppendToContainer/F_VN_AppendToContainer_TcVnVector2_DINT

	{attribute 'TcIecLibraryType'}
	{attribute 'external_name' := 'F_VN_AppendToContainer_TcVnVector2_DINT_GUID_DA320FEC_F72E_D1D3_A622_C9655E828B65'}
	(* Append a single element of type TcVnVector2_DINT to a container. *)
	FUNCTION F_VN_AppendToContainer_TcVnVector2_DINT : HRESULT
	VAR_IN_OUT
		aElement	:	TcVnVector2_DINT;	(* Single element to append to ipContainer *)
	END_VAR
	VAR_INPUT
		ipContainer	:	ITcVnContainer;	(* Container to which the element will be appended *)
		hrPrev	:	HRESULT;	(* HRESULT indicating the result of previous operations (If SUCCEEDED(hrPrev) equals false, no operation is executed.) *)
	END_VAR

END_FUNCTION

// Functions/Basic Container Operations/F_VN_AppendToContainer/F_VN_AppendToContainer_TcVnVector2_INT

	{attribute 'TcIecLibraryType'}
	{attribute 'external_name' := 'F_VN_AppendToContainer_TcVnVector2_INT_GUID_989841E8_475C_DF27_BEDA_634843ADB603'}
	(* Append a single element of type TcVnVector2_INT to a container. *)
	FUNCTION F_VN_AppendToContainer_TcVnVector2_INT : HRESULT
	VAR_IN_OUT
		aElement	:	TcVnVector2_INT;	(* Single element to append to ipContainer *)
	END_VAR
	VAR_INPUT
		ipContainer	:	ITcVnContainer;	(* Container to which the element will be appended *)
		hrPrev	:	HRESULT;	(* HRESULT indicating the result of previous operations (If SUCCEEDED(hrPrev) equals false, no operation is executed.) *)
	END_VAR

END_FUNCTION

// Functions/Basic Container Operations/F_VN_AppendToContainer/F_VN_AppendToContainer_TcVnVector2_REAL

	{attribute 'TcIecLibraryType'}
	{attribute 'external_name' := 'F_VN_AppendToContainer_TcVnVector2_REAL_GUID_512856B2_8488_D041_B821_D720B2904869'}
	(* Append a single element of type TcVnVector2_REAL to a container. *)
	FUNCTION F_VN_AppendToContainer_TcVnVector2_REAL : HRESULT
	VAR_IN_OUT
		aElement	:	TcVnVector2_REAL;	(* Single element to append to ipContainer *)
	END_VAR
	VAR_INPUT
		ipContainer	:	ITcVnContainer;	(* Container to which the element will be appended *)
		hrPrev	:	HRESULT;	(* HRESULT indicating the result of previous operations (If SUCCEEDED(hrPrev) equals false, no operation is executed.) *)
	END_VAR

END_FUNCTION

// Functions/Basic Container Operations/F_VN_AppendToContainer/F_VN_AppendToContainer_TcVnVector2_SINT

	{attribute 'TcIecLibraryType'}
	{attribute 'external_name' := 'F_VN_AppendToContainer_TcVnVector2_SINT_GUID_29C209E2_C3C8_DBD4_9948_895A996D9BE4'}
	(* Append a single element of type TcVnVector2_SINT to a container. *)
	FUNCTION F_VN_AppendToContainer_TcVnVector2_SINT : HRESULT
	VAR_IN_OUT
		aElement	:	TcVnVector2_SINT;	(* Single element to append to ipContainer *)
	END_VAR
	VAR_INPUT
		ipContainer	:	ITcVnContainer;	(* Container to which the element will be appended *)
		hrPrev	:	HRESULT;	(* HRESULT indicating the result of previous operations (If SUCCEEDED(hrPrev) equals false, no operation is executed.) *)
	END_VAR

END_FUNCTION

// Functions/Basic Container Operations/F_VN_AppendToContainer/F_VN_AppendToContainer_TcVnVector2_UINT

	{attribute 'TcIecLibraryType'}
	{attribute 'external_name' := 'F_VN_AppendToContainer_TcVnVector2_UINT_GUID_FE4BC28F_65C4_D819_ABBC_2A2404DA13E3'}
	(* Append a single element of type TcVnVector2_UINT to a container. *)
	FUNCTION F_VN_AppendToContainer_TcVnVector2_UINT : HRESULT
	VAR_IN_OUT
		aElement	:	TcVnVector2_UINT;	(* Single element to append to ipContainer *)
	END_VAR
	VAR_INPUT
		ipContainer	:	ITcVnContainer;	(* Container to which the element will be appended *)
		hrPrev	:	HRESULT;	(* HRESULT indicating the result of previous operations (If SUCCEEDED(hrPrev) equals false, no operation is executed.) *)
	END_VAR

END_FUNCTION

// Functions/Basic Container Operations/F_VN_AppendToContainer/F_VN_AppendToContainer_TcVnVector2_USINT

	{attribute 'TcIecLibraryType'}
	{attribute 'external_name' := 'F_VN_AppendToContainer_TcVnVector2_USINT_GUID_545F16C4_FB2B_DE57_A8EF_09C4026EE5FA'}
	(* Append a single element of type TcVnVector2_USINT to a container. *)
	FUNCTION F_VN_AppendToContainer_TcVnVector2_USINT : HRESULT
	VAR_IN_OUT
		aElement	:	TcVnVector2_USINT;	(* Single element to append to ipContainer *)
	END_VAR
	VAR_INPUT
		ipContainer	:	ITcVnContainer;	(* Container to which the element will be appended *)
		hrPrev	:	HRESULT;	(* HRESULT indicating the result of previous operations (If SUCCEEDED(hrPrev) equals false, no operation is executed.) *)
	END_VAR

END_FUNCTION

// Functions/Basic Container Operations/F_VN_AppendToContainer/F_VN_AppendToContainer_TcVnVector3_INT

	{attribute 'TcIecLibraryType'}
	{attribute 'external_name' := 'F_VN_AppendToContainer_TcVnVector3_INT_GUID_1DDF083F_93A0_D634_ADE3_157100112AB3'}
	(* Append a single element of type TcVnVector3_INT to a container. *)
	FUNCTION F_VN_AppendToContainer_TcVnVector3_INT : HRESULT
	VAR_IN_OUT
		aElement	:	TcVnVector3_INT;	(* Single element to append to ipContainer *)
	END_VAR
	VAR_INPUT
		ipContainer	:	ITcVnContainer;	(* Container to which the element will be appended *)
		hrPrev	:	HRESULT;	(* HRESULT indicating the result of previous operations (If SUCCEEDED(hrPrev) equals false, no operation is executed.) *)
	END_VAR

END_FUNCTION

// Functions/Basic Container Operations/F_VN_AppendToContainer/F_VN_AppendToContainer_TcVnVector3_REAL

	{attribute 'TcIecLibraryType'}
	{attribute 'external_name' := 'F_VN_AppendToContainer_TcVnVector3_REAL_GUID_494DBFF2_08D4_D66F_8859_F5E808F6D2EF'}
	(* Append a single element of type TcVnVector3_REAL to a container. *)
	FUNCTION F_VN_AppendToContainer_TcVnVector3_REAL : HRESULT
	VAR_IN_OUT
		aElement	:	TcVnVector3_REAL;	(* Single element to append to ipContainer *)
	END_VAR
	VAR_INPUT
		ipContainer	:	ITcVnContainer;	(* Container to which the element will be appended *)
		hrPrev	:	HRESULT;	(* HRESULT indicating the result of previous operations (If SUCCEEDED(hrPrev) equals false, no operation is executed.) *)
	END_VAR

END_FUNCTION

// Functions/Basic Container Operations/F_VN_AppendToContainer/F_VN_AppendToContainer_TcVnVector3_SINT

	{attribute 'TcIecLibraryType'}
	{attribute 'external_name' := 'F_VN_AppendToContainer_TcVnVector3_SINT_GUID_5B355138_7FCF_D45A_A119_AEC054F4CC5E'}
	(* Append a single element of type TcVnVector3_SINT to a container. *)
	FUNCTION F_VN_AppendToContainer_TcVnVector3_SINT : HRESULT
	VAR_IN_OUT
		aElement	:	TcVnVector3_SINT;	(* Single element to append to ipContainer *)
	END_VAR
	VAR_INPUT
		ipContainer	:	ITcVnContainer;	(* Container to which the element will be appended *)
		hrPrev	:	HRESULT;	(* HRESULT indicating the result of previous operations (If SUCCEEDED(hrPrev) equals false, no operation is executed.) *)
	END_VAR

END_FUNCTION

// Functions/Basic Container Operations/F_VN_AppendToContainer/F_VN_AppendToContainer_TcVnVector3_UINT

	{attribute 'TcIecLibraryType'}
	{attribute 'external_name' := 'F_VN_AppendToContainer_TcVnVector3_UINT_GUID_6D830F13_B4F2_D937_94B3_EB6854569671'}
	(* Append a single element of type TcVnVector3_UINT to a container. *)
	FUNCTION F_VN_AppendToContainer_TcVnVector3_UINT : HRESULT
	VAR_IN_OUT
		aElement	:	TcVnVector3_UINT;	(* Single element to append to ipContainer *)
	END_VAR
	VAR_INPUT
		ipContainer	:	ITcVnContainer;	(* Container to which the element will be appended *)
		hrPrev	:	HRESULT;	(* HRESULT indicating the result of previous operations (If SUCCEEDED(hrPrev) equals false, no operation is executed.) *)
	END_VAR

END_FUNCTION

// Functions/Basic Container Operations/F_VN_AppendToContainer/F_VN_AppendToContainer_TcVnVector3_USINT

	{attribute 'TcIecLibraryType'}
	{attribute 'external_name' := 'F_VN_AppendToContainer_TcVnVector3_USINT_GUID_10E3B7C3_59E3_D6EA_B8E4_A8AEAF9CE39D'}
	(* Append a single element of type TcVnVector3_USINT to a container. *)
	FUNCTION F_VN_AppendToContainer_TcVnVector3_USINT : HRESULT
	VAR_IN_OUT
		aElement	:	TcVnVector3_USINT;	(* Single element to append to ipContainer *)
	END_VAR
	VAR_INPUT
		ipContainer	:	ITcVnContainer;	(* Container to which the element will be appended *)
		hrPrev	:	HRESULT;	(* HRESULT indicating the result of previous operations (If SUCCEEDED(hrPrev) equals false, no operation is executed.) *)
	END_VAR

END_FUNCTION

// Functions/Basic Container Operations/F_VN_AppendToContainer/F_VN_AppendToContainer_TcVnVector4_DINT

	{attribute 'TcIecLibraryType'}
	{attribute 'external_name' := 'F_VN_AppendToContainer_TcVnVector4_DINT_GUID_1032A262_7E47_D8D9_A389_7981BED23D00'}
	(* Append a single element of type TcVnVector4_DINT to a container. *)
	FUNCTION F_VN_AppendToContainer_TcVnVector4_DINT : HRESULT
	VAR_IN_OUT
		aElement	:	TcVnVector4_DINT;	(* Single element to append to ipContainer *)
	END_VAR
	VAR_INPUT
		ipContainer	:	ITcVnContainer;	(* Container to which the element will be appended *)
		hrPrev	:	HRESULT;	(* HRESULT indicating the result of previous operations (If SUCCEEDED(hrPrev) equals false, no operation is executed.) *)
	END_VAR

END_FUNCTION

// Functions/Basic Container Operations/F_VN_AppendToContainer/F_VN_AppendToContainer_TcVnVector4_INT

	{attribute 'TcIecLibraryType'}
	{attribute 'external_name' := 'F_VN_AppendToContainer_TcVnVector4_INT_GUID_1B2F5F38_2B77_DD1A_A12F_A5EF27A9718E'}
	(* Append a single element of type TcVnVector4_INT to a container. *)
	FUNCTION F_VN_AppendToContainer_TcVnVector4_INT : HRESULT
	VAR_IN_OUT
		aElement	:	TcVnVector4_INT;	(* Single element to append to ipContainer *)
	END_VAR
	VAR_INPUT
		ipContainer	:	ITcVnContainer;	(* Container to which the element will be appended *)
		hrPrev	:	HRESULT;	(* HRESULT indicating the result of previous operations (If SUCCEEDED(hrPrev) equals false, no operation is executed.) *)
	END_VAR

END_FUNCTION

// Functions/Basic Container Operations/F_VN_AppendToContainer/F_VN_AppendToContainer_TcVnVector4_LREAL

	{attribute 'TcIecLibraryType'}
	{attribute 'external_name' := 'F_VN_AppendToContainer_TcVnVector4_LREAL_GUID_70107C7F_8B9A_DED1_AF97_9C8B55776AC2'}
	(* Append a single element of type TcVnVector4_LREAL to a container. *)
	FUNCTION F_VN_AppendToContainer_TcVnVector4_LREAL : HRESULT
	VAR_IN_OUT
		aElement	:	TcVnVector4_LREAL;	(* Single element to append to ipContainer *)
	END_VAR
	VAR_INPUT
		ipContainer	:	ITcVnContainer;	(* Container to which the element will be appended *)
		hrPrev	:	HRESULT;	(* HRESULT indicating the result of previous operations (If SUCCEEDED(hrPrev) equals false, no operation is executed.) *)
	END_VAR

END_FUNCTION

// Functions/Basic Container Operations/F_VN_AppendToContainer/F_VN_AppendToContainer_TcVnVector4_REAL

	{attribute 'TcIecLibraryType'}
	{attribute 'external_name' := 'F_VN_AppendToContainer_TcVnVector4_REAL_GUID_DBCF0703_D5D1_D7DA_BED9_BA1A6E8AD404'}
	(* Append a single element of type TcVnVector4_REAL to a container. *)
	FUNCTION F_VN_AppendToContainer_TcVnVector4_REAL : HRESULT
	VAR_IN_OUT
		aElement	:	TcVnVector4_REAL;	(* Single element to append to ipContainer *)
	END_VAR
	VAR_INPUT
		ipContainer	:	ITcVnContainer;	(* Container to which the element will be appended *)
		hrPrev	:	HRESULT;	(* HRESULT indicating the result of previous operations (If SUCCEEDED(hrPrev) equals false, no operation is executed.) *)
	END_VAR

END_FUNCTION

// Functions/Basic Container Operations/F_VN_AppendToContainer/F_VN_AppendToContainer_TcVnVector4_SINT

	{attribute 'TcIecLibraryType'}
	{attribute 'external_name' := 'F_VN_AppendToContainer_TcVnVector4_SINT_GUID_97C46AD7_821F_D134_ABD5_EDAB86731BDD'}
	(* Append a single element of type TcVnVector4_SINT to a container. *)
	FUNCTION F_VN_AppendToContainer_TcVnVector4_SINT : HRESULT
	VAR_IN_OUT
		aElement	:	TcVnVector4_SINT;	(* Single element to append to ipContainer *)
	END_VAR
	VAR_INPUT
		ipContainer	:	ITcVnContainer;	(* Container to which the element will be appended *)
		hrPrev	:	HRESULT;	(* HRESULT indicating the result of previous operations (If SUCCEEDED(hrPrev) equals false, no operation is executed.) *)
	END_VAR

END_FUNCTION

// Functions/Basic Container Operations/F_VN_AppendToContainer/F_VN_AppendToContainer_TcVnVector4_UINT

	{attribute 'TcIecLibraryType'}
	{attribute 'external_name' := 'F_VN_AppendToContainer_TcVnVector4_UINT_GUID_9BB38CBC_835D_D6C6_92AD_F86492768E4C'}
	(* Append a single element of type TcVnVector4_UINT to a container. *)
	FUNCTION F_VN_AppendToContainer_TcVnVector4_UINT : HRESULT
	VAR_IN_OUT
		aElement	:	TcVnVector4_UINT;	(* Single element to append to ipContainer *)
	END_VAR
	VAR_INPUT
		ipContainer	:	ITcVnContainer;	(* Container to which the element will be appended *)
		hrPrev	:	HRESULT;	(* HRESULT indicating the result of previous operations (If SUCCEEDED(hrPrev) equals false, no operation is executed.) *)
	END_VAR

END_FUNCTION

// Functions/Basic Container Operations/F_VN_AppendToContainer/F_VN_AppendToContainer_TcVnVector4_USINT

	{attribute 'TcIecLibraryType'}
	{attribute 'external_name' := 'F_VN_AppendToContainer_TcVnVector4_USINT_GUID_778A40D1_6733_DB85_852B_17C8E7A614B2'}
	(* Append a single element of type TcVnVector4_USINT to a container. *)
	FUNCTION F_VN_AppendToContainer_TcVnVector4_USINT : HRESULT
	VAR_IN_OUT
		aElement	:	TcVnVector4_USINT;	(* Single element to append to ipContainer *)
	END_VAR
	VAR_INPUT
		ipContainer	:	ITcVnContainer;	(* Container to which the element will be appended *)
		hrPrev	:	HRESULT;	(* HRESULT indicating the result of previous operations (If SUCCEEDED(hrPrev) equals false, no operation is executed.) *)
	END_VAR

END_FUNCTION

// Functions/Basic Container Operations/F_VN_AppendToContainer/F_VN_AppendToContainer_UDINT

	{attribute 'TcIecLibraryType'}
	{attribute 'external_name' := 'F_VN_AppendToContainer_UDINT_GUID_9C7D5416_9EC1_D40F_9FA1_77AF30CEA8BE'}
	(* Append a single element of type UDINT to a container. *)
	FUNCTION F_VN_AppendToContainer_UDINT : HRESULT
	VAR_INPUT
		nElement	:	UDINT;	(* Single element to append to ipContainer *)
		ipContainer	:	ITcVnContainer;	(* Container to which the element will be appended *)
		hrPrev	:	HRESULT;	(* HRESULT indicating the result of previous operations (If SUCCEEDED(hrPrev) equals false, no operation is executed.) *)
	END_VAR

END_FUNCTION

// Functions/Basic Container Operations/F_VN_AppendToContainer/F_VN_AppendToContainer_UINT

	{attribute 'TcIecLibraryType'}
	{attribute 'external_name' := 'F_VN_AppendToContainer_UINT_GUID_263616FE_D5A6_D3EA_A903_2FF330F999D0'}
	(* Append a single element of type UINT to a container. *)
	FUNCTION F_VN_AppendToContainer_UINT : HRESULT
	VAR_INPUT
		nElement	:	UINT;	(* Single element to append to ipContainer *)
		ipContainer	:	ITcVnContainer;	(* Container to which the element will be appended *)
		hrPrev	:	HRESULT;	(* HRESULT indicating the result of previous operations (If SUCCEEDED(hrPrev) equals false, no operation is executed.) *)
	END_VAR

END_FUNCTION

// Functions/Basic Container Operations/F_VN_AppendToContainer/F_VN_AppendToContainer_ULINT

	{attribute 'TcIecLibraryType'}
	{attribute 'external_name' := 'F_VN_AppendToContainer_ULINT_GUID_AA2B082D_F9D7_D0A1_AA2C_7A7A708FABE3'}
	(* Append a single element of type ULINT to a container. *)
	FUNCTION F_VN_AppendToContainer_ULINT : HRESULT
	VAR_INPUT
		nElement	:	ULINT;	(* Single element to append to ipContainer *)
		ipContainer	:	ITcVnContainer;	(* Container to which the element will be appended *)
		hrPrev	:	HRESULT;	(* HRESULT indicating the result of previous operations (If SUCCEEDED(hrPrev) equals false, no operation is executed.) *)
	END_VAR

END_FUNCTION

// Functions/Basic Container Operations/F_VN_AppendToContainer/F_VN_AppendToContainer_USINT

	{attribute 'TcIecLibraryType'}
	{attribute 'external_name' := 'F_VN_AppendToContainer_USINT_GUID_14AC29BC_1C52_D7B9_B544_A5F970141C96'}
	(* Append a single element of type USINT to a container. *)
	FUNCTION F_VN_AppendToContainer_USINT : HRESULT
	VAR_INPUT
		nElement	:	USINT;	(* Single element to append to ipContainer *)
		ipContainer	:	ITcVnContainer;	(* Container to which the element will be appended *)
		hrPrev	:	HRESULT;	(* HRESULT indicating the result of previous operations (If SUCCEEDED(hrPrev) equals false, no operation is executed.) *)
	END_VAR

END_FUNCTION

// Functions/Basic Container Operations/F_VN_FillContainer/F_VN_FillContainer_DINT

	{attribute 'TcIecLibraryType'}
	{attribute 'external_name' := 'F_VN_FillContainer_DINT_GUID_10332741_CCDA_D28D_BEF5_6ED5C1214FB8'}
	(* Fill the container with the specified value. Only possible for containers with basic elements. *)
	FUNCTION F_VN_FillContainer_DINT : HRESULT
	VAR_INPUT
		ipContainer	:	ITcVnContainer;	(* Container with basic elements *)
		nValue	:	DINT;	(* Value to set the container elements *)
		hrPrev	:	HRESULT;	(* HRESULT indicating the result of previous operations (If SUCCEEDED(hrPrev) equals false, no operation is executed.) *)
	END_VAR

END_FUNCTION

// Functions/Basic Container Operations/F_VN_FillContainer/F_VN_FillContainer_INT

	{attribute 'TcIecLibraryType'}
	{attribute 'external_name' := 'F_VN_FillContainer_INT_GUID_96DEAA40_3290_D7EE_A789_4B241D79A647'}
	(* Fill the container with the specified value. Only possible for containers with basic elements. *)
	FUNCTION F_VN_FillContainer_INT : HRESULT
	VAR_INPUT
		ipContainer	:	ITcVnContainer;	(* Container with basic elements *)
		nValue	:	INT;	(* Value to set the container elements *)
		hrPrev	:	HRESULT;	(* HRESULT indicating the result of previous operations (If SUCCEEDED(hrPrev) equals false, no operation is executed.) *)
	END_VAR

END_FUNCTION

// Functions/Basic Container Operations/F_VN_FillContainer/F_VN_FillContainer_ITcVnImage

